		IF (left_groud_check1 AND left_groud_check2) THEN
			IF(head_f2 )THEN  ton_step4(in:=TRUE,pt:=T#1.5s);
			ELSE IF(head_b2 )THEN  ton_step4(in:=TRUE,pt:=T#1.0s);
			ELSE IF(head_b)THEN ton_step4(in:=TRUE,pt:=T#1.0s);
			ELSE IF(head_f)THEN ton_step4(in:=TRUE,pt:=T#2.0s);
			ELSE 	ton_step4(in:=TRUE,pt:=T#2.0s);
			END_IF
			END_IF
			END_IF
			END_IF
		END_IF


		IF ton1.q THEN leave_ground_sign:=1;ELSE leave_ground_sign:=0;END_IF
		IF( (ton_step4.q OR ton1.q )AND NOT level_second )OR (level_second AND ton4_second.Q )OR ton6_yanshi.Q THEN
			ton_step4(in:=0);
			ton1(in:=0);
			ton4_second(in:=0);
			extend_step:=5;
			step4_m1:=0;
			step4_m2:=0;
			step4_m3:=0;
			step4_m4:=0;
		END_IF
	END_IF

(*————————————————————————————自动支腿第五步————————————————————————————————————————*)
(*控制过程：精调平*)
	IF extend_step = 5 THEN
		tem2:=INT_TO_DINT(level_time)*1000;
		ton1(in:=1,pt:=DINT_TO_TIME(tem2));

		ton1();
		angle_x_real:=INT_TO_REAL(angle_x);
		angle_x_offset_real:=INT_TO_REAL(angle_x_offset);
		set_x:=REAL_TO_WORD(ABS(angle_x_real-angle_x_offset_real));
		angle_y_real:=INT_TO_REAL(angle_y);
		angle_y_offset_real:=INT_TO_REAL(angle_y_offset);
		set_y:=REAL_TO_WORD(ABS(angle_y_real-angle_y_offset_real));set_y := set_y*8/rl_ys;
		angle_ok_sign:=angle_ok/2;
		 IF REAL_TO_INT(ABS(angle_x_real-angle_x_offset_real)) <= angle_ok_sign THEN set_x := 0; END_IF;
		 IF REAL_TO_INT(ABS(angle_y_real-angle_y_offset_real)) <= angle_ok_sign THEN set_y := 0; END_IF;
(*--------------------------------------------------*)
		IF (angle_x-angle_x_offset)>=angle_ok_sign AND (angle_y-angle_y_offset)<=angle_ok_sign THEN
				left_front_desired:=set_x;
				right_back_desired:=set_y;
				left_back_desired:=set_x+set_y;
			IF NOT back_left_urt_ex_check THEN
				left_back_desired:=left_back_desired*2;left_front_desired:=left_front_desired/2;	right_back_desired:=right_back_desired/2;
    			END_IF
		ELSIF (angle_x-angle_x_offset)>=angle_ok_sign AND (angle_y-angle_y_offset)>=angle_ok_sign THEN
(*				right_front_desired:=set_y;*)
				left_back_desired:=set_x;
				left_front_desired:=set_x+set_y;
			IF NOT front_left_urt_ex_check THEN
				left_front_desired:=left_front_desired*2;	left_back_desired:=left_back_desired/2;	right_front_desired:=right_front_desired/2;
    			END_IF
		ELSIF (angle_x-angle_x_offset)<=angle_ok_sign AND (angle_y-angle_y_offset)<=angle_ok_sign THEN
				left_back_desired:=set_y;
				right_front_desired:=set_x;
				right_back_desired:=set_x+set_y;
			IF NOT back_right_urt_ex_check THEN
				right_back_desired:=right_back_desired*2;
				left_back_desired:=left_back_desired/2;
				right_front_desired:=right_front_desired/2;
    			END_IF
		ELSIF (angle_x-angle_x_offset)<=angle_ok_sign AND (angle_y-angle_y_offset)>=angle_ok_sign THEN
				right_back_desired:=set_x;
(*				left_front_desired:=set_y;*)
				right_front_desired:=set_x+set_y;
			IF NOT front_right_urt_ex_check THEN
				right_front_desired:=right_front_desired*2;	right_back_desired:=right_back_desired/2;	left_front_desired:=left_front_desired/2;
   			END_IF
		END_IF
(*************sl 增加******************s*)
			IF(head_b AND (angle_y>angle_y_offset))THEN
				IF(angle_x>angle_x_offset)THEN
						left_front_desired:=left_front_desired+20;
						right_front_desired:=right_front_desired+15;
						 left_back_desired:=REAL_TO_WORD(WORD_TO_REAL(left_back_desired)-5);
						 right_back_desired:=REAL_TO_WORD(WORD_TO_REAL(right_back_desired)-10);
				END_IF
				IF(angle_x<angle_x_offset)THEN
						left_front_desired:=left_front_desired+15;
						right_front_desired:=right_front_desired+20;
						left_back_desired:=REAL_TO_WORD(WORD_TO_REAL(left_back_desired)-10);
						 right_back_desired:=REAL_TO_WORD(WORD_TO_REAL(right_back_desired)-5);
				END_IF
			END_IF

			IF(head_f AND (angle_y<angle_y_offset))THEN
				IF(angle_x>angle_x_offset)THEN
						left_front_desired:=REAL_TO_WORD(WORD_TO_REAL(left_front_desired)-5);
						 right_front_desired:=REAL_TO_WORD(WORD_TO_REAL(right_front_desired)-10);
						left_back_desired:=left_back_desired+20;
						right_back_desired:=right_back_desired+15;
				END_IF
				IF(angle_x<angle_x_offset)THEN
						left_front_desired:=REAL_TO_WORD(WORD_TO_REAL(left_front_desired)-10);
						 right_front_desired:=REAL_TO_WORD(WORD_TO_REAL(right_front_desired)-5);
						left_back_desired:=left_back_desired+15;
						right_back_desired:=right_back_desired+20;
				END_IF
			END_IF
(*************sl 增加******************e*)
		IF NOT front_left_urt_ex_check1  THEN left_front_desired:=300;END_IF
		IF NOT back_left_urt_ex_check1   THEN  left_back_desired:=300;END_IF
		IF NOT front_right_urt_ex_check1 THEN   right_front_desired:=300;END_IF
		IF NOT back_right_urt_ex_check1 THEN  right_back_desired:=300;END_IF

IF (angle_y-angle_y_offset)<-step_4_limit+100 THEN left_front_desired:=0;right_front_desired:=0;END_IF
IF (angle_y-angle_y_offset)>step_4_limit-100 THEN right_back_desired:=0;left_back_desired:=0;END_IF
IF (angle_x-angle_x_offset)<-step_4_limit+100 THEN left_front_desired:=0;left_back_desired:=0;END_IF
IF (angle_x-angle_x_offset)>step_4_limit-100 THEN right_back_desired:=0;right_front_desired:=0;END_IF
		tontp(IN:= ABS(angle_x-angle_x_offset)<=angle_ok AND ABS(angle_y-angle_y_offset)<=angle_ok, PT:= T#200ms);
  (*精调平完成*)
		IF front_left_urt_ex_check AND front_right_urt_ex_check AND back_right_urt_ex_check AND back_left_urt_ex_check
			AND tontp.Q AND(( left_groud_check1 AND left_groud_check2)OR ton6_yanshi.Q  )THEN
(*			extend_do := 0;*)			ton1(in:=0);			(*leveled := 1;*)		alarmer_horn:=0;
			extend_step:=7;			down_valve_ctl:=0;
		END_IF;
		IF NOT(left_groud_check1 AND left_groud_check2)AND NOT ton6_yanshi.Q  THEN extend_step := 4; END_IF; (*有轮胎触地，回到撑起步骤*)
		IF ton1.q THEN ton1(in:=0); extend_step:=6;END_IF
	END_IF
(*————————————————————————————自动支腿第六步————————————————————————————————————————*)
	IF extend_step=6 THEN
		left_back_drawback_desired:=v_in_speed;
		left_front_drawback_desired:=v_in_speed;
		right_back_drawback_desired:=v_in_speed;
		right_front_drawback_desired:=v_in_speed;
		IF (NOT ton6_yanshi.Q AND (NOT left_groud_check1 OR NOT left_groud_check2)) OR
			NOT(front_left_urt_ex_check AND front_right_urt_ex_check AND back_left_urt_ex_check AND back_right_urt_ex_check) THEN
			extend_step:=4;
			ton6_yanshi(in:=0);
		END_IF
	END_IF

IF left_front_desired<0 OR  left_front_desired>10000 			THEN left_front_desired:=0;END_IF
IF left_back_desired<0 OR  left_back_desired>10000		 	THEN left_back_desired:=0;END_IF
IF right_front_desired<0 OR  right_front_desired>10000 		THEN right_front_desired:=0;END_IF
IF right_back_desired<0 OR  right_back_desired>10000		 THEN right_back_desired:=0;END_IF

(************************************伸支腿后展斗****************************************s*)
	stage_extend_do:=1;
	stage_draw_do:=0;

IF extend_step=7 THEN
	down_valve_ctl:=0;
	up_valve_ctl:=0;
	IF stage_extend_over THEN
		extend_do := 0;
		extend_step:=0;
		leveled := 1;
		alarmer_horn:=0;
		stage_extend_do:=0;
		stage_extend_over:=0;
	END_IF
END_IF
(************************************伸支腿后展斗****************************************e*)
ELSE
	extend_step:=0;
	stage_extend_do:=0;
	leave_ground_sign:=0;
END_IF



(*sl*****************************非正常调平判定*******************start*)
(**)
IF NOT auto_manu_choice AND((front_right_Lv_ex_check AND back_right_Lv_ex_check)OR(front_left_Lv_ex_check AND back_left_Lv_ex_check))AND front_left_urt_ex_check AND front_right_urt_ex_check AND back_left_urt_ex_check AND back_right_urt_ex_check AND ABS(angle_x-angle_x_offset)<=1.5*angle_ok AND ABS(angle_y-angle_y_offset)<=1.5*angle_ok THEN
	leveled:=1;
END_IF

(*sl*****************************非正常调平判定*******************end*)
(*
ton_second(in:=1,pt:=t#15s);
IF ton_second.Q  THEN allow_second:=1; END_IF
IF allow_second THEN
*)

(*
	IF NOT(front_left_urt_ex_check OR front_right_urt_ex_check OR back_left_urt_ex_check OR back_right_urt_ex_check)  AND  valve_act THEN
		leveled:=0;
	END_IF
ton_second()
*)
IF NOT(front_left_urt_ex_check OR front_right_urt_ex_check OR back_left_urt_ex_check OR back_right_urt_ex_check)  AND  valve_act THEN
	allow_second:=1;
ELSE
	allow_second:=0;
END_IF
ton_second(in:=allow_second,pt:=t#2s);
IF ton_second.Q THEN 		leveled:=0; 	ton_second(in:=0);	END_IF

(*————————————————————————————收支腿————————————————————————————————————————*)
(*收回支腿操作*)
auto_drawback_triger:=auto_drawback_triger_left OR auto_drawback_triger_right;
drawback_act(CLK:= auto_drawback_triger);
(*臂架到位而且不是第二次按收回旋钮*)
IF drawback_act.q  AND arm_to_station AND auto_manu_choice THEN
	withdraw_do:=(NOT withdraw_do);
	leave_ground_sign:=0;
	extend_do:=0;
	ton1(in:=0);ton6_yanshi(in:=0);
	withdraw_step:=100;
END_IF


(************************************收支腿前翻斗****************************************e*)

(*收回步骤1：收垂直腿*)
IF withdraw_do THEN

(************************************收支腿前翻斗****************************************s*)
(*
IF withdraw_step=10 THEN
	stage_extend_do:=0;
	stage_draw_do:=1;
	down_valve_ctl:=0;
	up_valve_ctl:=1;
	IF stage_draw_over THEN
		withdraw_step:=100;
		stage_draw_do:=0;
		stage_draw_over:=0;
	END_IF
ELSE
	stage_draw_do:=0;
END_IF
*)
stage_extend_do:=0;
stage_draw_do:=1;
IF stage_draw_over THEN
	stage_draw_do:=0;
	stage_draw_over:=0;
END_IF


IF withdraw_step=100 THEN
	ton_withdraw(in:=1,pt:=t#1s);
	IF(ton_withdraw.Q)THEN
		withdraw_step:=1;
		ton_withdraw(in:=0);
	END_IF
END_IF

	alarmer_horn:=1;

	IF withdraw_step=1 THEN
		tem2:=INT_TO_DINT(v_in_time)*1000;
		ton1(in:=1,pt:=DINT_TO_TIME(tem2));
		ton1();
		IF NOT front_left_urt_drb_check 		THEN left_front_drawback_desired:=v_in_speed; 	ELSE	left_front_drawback_desired:=0;		END_IF
		IF NOT front_right_urt_drb_check 	THEN right_front_drawback_desired:=v_in_speed;	ELSE	right_front_drawback_desired:=0; 	END_IF
		IF NOT back_left_urt_drb_check 		THEN left_back_drawback_desired:=v_in_speed; 	ELSE	left_back_drawback_desired:=0;		END_IF
		IF NOT back_right_urt_drb_check	THEN right_back_drawback_desired:=v_in_speed; ELSE	right_back_drawback_desired:=0;	END_IF

(*************sl 增加******************s*结合象限角结合XY变化率来对速度开口进行加减*)
IF(NOT  left_groud_check1 AND NOT  left_groud_check2)THEN
	withdraw_t1(in:=1,pt:=t#2s);
	IF(withdraw_t1.Q)THEN
		withdraw_m5:=1;
	END_IF
END_IF

IF(NOT withdraw_m5 )OR(head_b2 AND(back_right_urt_ex_check OR back_left_urt_ex_check))OR(head_f2 AND(front_right_urt_ex_check OR front_left_urt_ex_check))THEN
	IF  NOT( angle_withdraw_x1=angle_x )THEN
		angle_withdraw_x2:=angle_withdraw_x1;
		angle_withdraw_x1:=angle_x;
	END_IF
	IF  NOT( angle_withdraw_y1=angle_y )THEN
		angle_withdraw_y2:=angle_withdraw_y1;
		angle_withdraw_y1:=angle_y;
	END_IF
	withdraw_mx:=angle_withdraw_x1-angle_withdraw_x2;
	withdraw_my:=angle_withdraw_y1-angle_withdraw_y2;

	CASE angle_dir OF(*清零 以及 各项先+-50*)
		1:
			withdraw_m1:=1;
			IF(withdraw_m2 OR withdraw_m3 OR withdraw_m4)THEN
				withdraw_fl:=0;
				withdraw_fr:=0;
				withdraw_bl:=0;
				withdraw_br:=0;
				withdraw_m2:=0;withdraw_m3:=0;withdraw_m4:=0;
			END_IF
			IF(angle_x>=angle_x_offset+50)THEN
				IF(withdraw_mx>0)THEN withdraw_fr:=withdraw_fr+w_value; withdraw_br:=withdraw_br+w_value;   END_IF
			END_IF
			IF(angle_y<=angle_y_offset-50)THEN
				 withdraw_fl:=withdraw_fl+w_value;  withdraw_fr:=withdraw_fr+w_value;
			END_IF
			IF(withdraw_my<0)THEN
				withdraw_fl:=withdraw_fl+w_value;  withdraw_fr:=withdraw_fr+w_value;
			END_IF

		2:
			withdraw_m2:=1;
			IF(withdraw_m1 OR withdraw_m3 OR withdraw_m4)THEN
				withdraw_fl:=0;
				withdraw_fr:=0;
				withdraw_bl:=0;
				withdraw_br:=0;
				withdraw_m1:=0;withdraw_m3:=0;withdraw_m4:=0;
			END_IF
			IF(angle_x>=angle_x_offset+50)THEN
				IF(withdraw_mx>0)THEN withdraw_fr:=withdraw_fr+w_value; withdraw_br:=withdraw_br+w_value;   END_IF
			END_IF
			IF(angle_y>=angle_y_offset+50)THEN
				 withdraw_bl:=withdraw_bl+w_value;  withdraw_br:=withdraw_br+w_value;
			END_IF
			IF(withdraw_my>0)THEN
				withdraw_bl:=withdraw_bl+w_value;  withdraw_br:=withdraw_br+w_value;
			END_IF
		3:
			withdraw_m3:=1;
			IF(withdraw_m2 OR withdraw_m1 OR withdraw_m4)THEN
				withdraw_fl:=0;
				withdraw_fr:=0;
				withdraw_bl:=0;
				withdraw_br:=0;
				withdraw_m1:=0;withdraw_m2:=0;withdraw_m4:=0;
			END_IF
			IF(angle_x<=angle_x_offset-50)THEN
				IF(withdraw_mx<0)THEN withdraw_fl:=withdraw_fl+w_value; withdraw_bl:=withdraw_bl+w_value;   END_IF
			END_IF
			IF(angle_y<=angle_y_offset-50)THEN
				 withdraw_fl:=withdraw_fl+w_value;  withdraw_fr:=withdraw_fr+w_value;
			END_IF
			IF(withdraw_my<0)THEN
				withdraw_fl:=withdraw_fl+w_value;  withdraw_fr:=withdraw_fr+w_value;
			END_IF
		4:
			withdraw_m4:=1;
			IF(withdraw_m2 OR withdraw_m3 OR withdraw_m1)THEN
				withdraw_fl:=0;
				withdraw_fr:=0;
				withdraw_bl:=0;
				withdraw_br:=0;
				withdraw_m1:=0;withdraw_m2:=0;withdraw_m3:=0;
			END_IF
			IF(angle_x<=angle_x_offset-50)THEN
				IF(withdraw_mx<0)THEN withdraw_fl:=withdraw_fl+w_value; withdraw_bl:=withdraw_bl+w_value;   		END_IF
			END_IF
			IF(angle_y>=angle_y_offset+50)THEN
				withdraw_bl:=withdraw_bl+w_value;  withdraw_br:=withdraw_br+w_value;
			END_IF
			IF(withdraw_my>0)THEN
				withdraw_bl:=withdraw_bl+w_value;  withdraw_br:=withdraw_br+w_value;
			END_IF
	END_CASE

		IF NOT front_left_urt_drb_check 		THEN left_front_drawback_desired:=v_in_speed-withdraw_fl; 			ELSE	left_front_drawback_desired:=0;		END_IF
		IF NOT front_right_urt_drb_check 	THEN right_front_drawback_desired:=v_in_speed-withdraw_fr;		ELSE	right_front_drawback_desired:=0; 	END_IF
		IF NOT back_left_urt_drb_check 		THEN left_back_drawback_desired:=v_in_speed-withdraw_bl; 		ELSE	left_back_drawback_desired:=0;		END_IF
		IF NOT back_right_urt_drb_check	THEN right_back_drawback_desired:=v_in_speed-withdraw_br;	 	ELSE	right_back_drawback_desired:=0;	END_IF
ELSE
		withdraw_fl:=0;
		withdraw_fr:=0;
		withdraw_bl:=0;
		withdraw_br:=0;
END_IF
(*************sl 增加******************e*)

		IF (front_left_urt_drb_check AND front_right_urt_drb_check AND back_left_urt_drb_check AND back_right_urt_drb_check)OR ton1.q THEN
		ton1(in:=0);
		withdraw_t1(in:=0);
		withdraw_step:=2;
		withdraw_m5:=0;
		END_IF

	END_IF
	IF withdraw_step=2 THEN

		tem2:=INT_TO_DINT(v_in_time)*1000;
		ton1(in:=1,pt:=DINT_TO_TIME(tem2));
		ton1();
		IF NOT front_left_Lv_drb_check  	THEN left_front_lv_drb_valve:=1;   	ELSE	left_front_lv_drb_valve:=0;	END_IF
		IF NOT back_left_lv_drb_check   	THEN left_back_lv_drb_valve:=1;		ELSE	left_back_lv_drb_valve:=0; 	END_IF
		IF NOT front_right_lv_drb_check 	THEN right_front_lv_drb_valve:=1; 	ELSE	right_front_lv_drb_valve:=0;	END_IF
		IF NOT back_right_lv_drb_check  THEN right_back_lv_drb_valve:=1; 	ELSE	right_back_lv_drb_valve:=0;	END_IF
		IF ((front_left_Lv_drb_check AND back_left_lv_drb_check AND front_right_lv_drb_check AND back_right_lv_drb_check) OR ton1.q )AND NOT stage_draw_do THEN
			ton1(in:=0);
			withdraw_do:=0;
			withdraw_step:=0;
			down_valve_ctl:=0;
			up_valve_ctl:=0;
			head_f:=0;head_b:=0;head_f2:=0;head_b2:=0;side_l:=0;side_r:=0;
		END_IF
END_IF
	IF NOT front_left_urt_drb_check 		THEN left_front_drawback_desired:=v_in_speed; 	ELSE	left_front_drawback_desired:=0;				END_IF
			IF NOT front_right_urt_drb_check 	THEN right_front_drawback_desired:=v_in_speed;	ELSE	right_front_drawback_desired:=0; 	END_IF
			IF NOT back_left_urt_drb_check 		THEN left_back_drawback_desired:=v_in_speed; 	ELSE	left_back_drawback_desired:=0;		END_IF
			IF NOT back_right_urt_drb_check	THEN right_back_drawback_desired:=v_in_speed; ELSE	right_back_drawback_desired:=0;	END_IF
	END_IF

IF withdraw_do THEN
	leveled:=0;
ELSE
	withdraw_step:=0;
	stage_draw_do:=0;
END_IF
END_PROGRAM

(* POU TRIGER_Regulation/LEVEL_PROMPT, ST *)
PROGRAM LEVEL_PROMPT
VAR
	left_front_desired_prom_add1: BOOL;
	R_TRIG1: R_TRIG;
	R_TRIG2: R_TRIG;
	R_TRIG3: R_TRIG;
	R_TRIG4: R_TRIG;
	R_TRIG5: R_TRIG;
	R_TRIG6: R_TRIG;
	R_TRIG7: R_TRIG;
	R_TRIG8: R_TRIG;


	R_TRIG9: R_TRIG;
	R_TRIG10: R_TRIG;
	R_TRIG11: R_TRIG;
	R_TRIG12: R_TRIG;
	R_TRIG13: R_TRIG;
	R_TRIG14: R_TRIG;
	R_TRIG15: R_TRIG;
	R_TRIG16: R_TRIG;


	R_TRIG17: R_TRIG;
	R_TRIG18: R_TRIG;
	R_TRIG19: R_TRIG;
	R_TRIG20: R_TRIG;
	R_TRIG21: R_TRIG;
	R_TRIG22: R_TRIG;
	R_TRIG23: R_TRIG;
	R_TRIG24: R_TRIG;

	fl_o_fac_b1: BOOL;
	fr_o_fac_b1: BOOL;
	rl_o_fac_b1: BOOL;
	rr_o_fac_b1: BOOL;
	fl_i_fac_b1: BOOL;
	fr_i_fac_b1: BOOL;
	rl_i_fac_b1: BOOL;
	rr_i_fac_b1: BOOL;

	fl_o_fac_b_l1: BOOL;
	fr_o_fac_b_l1: BOOL;
	rl_o_fac_b_l1: BOOL;
	rr_o_fac_b_l1: BOOL;
	fl_i_fac_b_l1: BOOL;
	fr_i_fac_b_l1: BOOL;
	rl_i_fac_b_l1: BOOL;
	rr_i_fac_b_l1: BOOL;

	fl_o_fac_b_r1: BOOL;
	fr_o_fac_b_r1: BOOL;
	rl_o_fac_b_r1: BOOL;
	rr_o_fac_b_r1: BOOL;
	fl_i_fac_b_r1: BOOL;
	fr_i_fac_b_r1: BOOL;
	rl_i_fac_b_r1: BOOL;
	rr_i_fac_b_r1: BOOL;


END_VAR
digit_data_in_cylinder();

IF(head_b2)OR(head_f2)THEN
	case_curve2();
ELSE
	case_curve();
END_IF


IF NOT ramp_selected THEN

	analog_in_out_cylinder();

	R_TRIG1(CLK:=fl_o_fac_b , Q=>fl_o_fac_b1 );
	R_TRIG2(CLK:=fl_i_fac_b , Q=>fl_i_fac_b1 );
	IF fl_o_fac_b1 THEN fl_fac_nr:=fl_fac_nr+1;END_IF
	IF fl_i_fac_b1 THEN fl_fac_nr:=fl_fac_nr-1;END_IF
	IF fl_fac_nr>10 THEN fl_fac_nr:=10;END_IF
	IF fl_fac_nr<-10 THEN fl_fac_nr:=-10;END_IF

	R_TRIG3(CLK:=fl_o_fac_b_l , Q=>fl_o_fac_b_l1 );
	R_TRIG4(CLK:=fl_i_fac_b_l , Q=>fl_i_fac_b_l1 );
	IF fl_o_fac_b_l1 THEN fl_fac_l_nr:=fl_fac_l_nr+1;END_IF
	IF fl_i_fac_b_l1 THEN fl_fac_l_nr:=fl_fac_l_nr-1;END_IF
	IF fl_fac_l_nr>10 THEN fl_fac_l_nr:=10;END_IF
	IF fl_fac_l_nr<-10 THEN fl_fac_l_nr:=-10;END_IF

	R_TRIG5(CLK:=fl_o_fac_b_r , Q=>fl_o_fac_b_r1 );
	R_TRIG6(CLK:=fl_i_fac_b_r , Q=>fl_i_fac_b_r1 );
	IF fl_o_fac_b_r1 THEN fl_fac_r_nr:=fl_fac_r_nr+1;END_IF
	IF fl_i_fac_b_r1 THEN fl_fac_r_nr:=fl_fac_r_nr-1;END_IF
	IF fl_fac_r_nr>10 THEN fl_fac_r_nr:=10;END_IF
	IF fl_fac_r_nr<-10 THEN fl_fac_r_nr:=-10;END_IF
	(***********************************)

	R_TRIG7(CLK:=fr_o_fac_b , Q=>fr_o_fac_b1 );
	R_TRIG8(CLK:=fr_i_fac_b , Q=>fr_i_fac_b1 );
	IF fr_o_fac_b1 THEN fr_fac_nr:=fr_fac_nr+1;END_IF
	IF fr_i_fac_b1 THEN fr_fac_nr:=fr_fac_nr-1;END_IF
	IF fr_fac_nr>10 THEN fr_fac_nr:=10;END_IF
	IF fr_fac_nr<-10 THEN fr_fac_nr:=-10;END_IF

	R_TRIG9(CLK:=fr_o_fac_b_l , Q=>fr_o_fac_b_l1 );
	R_TRIG10(CLK:=fr_i_fac_b_l , Q=>fr_i_fac_b_l1 );
	IF fr_o_fac_b_l1 THEN fr_fac_l_nr:=fr_fac_l_nr+1;END_IF
	IF fr_i_fac_b_l1 THEN fr_fac_l_nr:=fr_fac_l_nr-1;END_IF
	IF fr_fac_l_nr>10 THEN fr_fac_l_nr:=10;END_IF
	IF fr_fac_l_nr<-10 THEN fr_fac_l_nr:=-10;END_IF

	R_TRIG11(CLK:=fr_o_fac_b_r , Q=>fr_o_fac_b_r1 );
	R_TRIG12(CLK:=fr_i_fac_b_r , Q=>fr_i_fac_b_r1 );
	IF fr_o_fac_b_r1 THEN fr_fac_r_nr:=fr_fac_r_nr+1;END_IF
	IF fr_i_fac_b_r1 THEN fr_fac_r_nr:=fr_fac_r_nr-1;END_IF
	IF fr_fac_r_nr>10 THEN fr_fac_r_nr:=10;END_IF
	IF fr_fac_r_nr<-10 THEN fr_fac_r_nr:=-10;END_IF

	(*******************************)

	R_TRIG13(CLK:=rl_o_fac_b , Q=>rl_o_fac_b1 );
	R_TRIG14(CLK:=rl_i_fac_b , Q=>rl_i_fac_b1 );
	IF rl_o_fac_b1 THEN rl_fac_nr:=rl_fac_nr+1;END_IF
	IF rl_i_fac_b1 THEN rl_fac_nr:=rl_fac_nr-1;END_IF
	IF rl_fac_nr>10 THEN rl_fac_nr:=10;END_IF
	IF rl_fac_nr<-10 THEN rl_fac_nr:=-10;END_IF

	R_TRIG15(CLK:=rl_o_fac_b_l , Q=>rl_o_fac_b_l1 );
	R_TRIG16(CLK:=rl_i_fac_b_l , Q=>rl_i_fac_b_l1 );
	IF rl_o_fac_b_l1 THEN rl_fac_l_nr:=rl_fac_l_nr+1;END_IF
	IF rl_i_fac_b_l1 THEN rl_fac_l_nr:=rl_fac_l_nr-1;END_IF
	IF rl_fac_l_nr>10 THEN rl_fac_l_nr:=10;END_IF
	IF rl_fac_l_nr<-10 THEN rl_fac_l_nr:=-10;END_IF

	R_TRIG17(CLK:=rl_o_fac_b_r , Q=>rl_o_fac_b_r1 );
	R_TRIG18(CLK:=rl_i_fac_b_r , Q=>rl_i_fac_b_r1 );
	IF rl_o_fac_b_r1 THEN rl_fac_r_nr:=rl_fac_r_nr+1;END_IF
	IF rl_i_fac_b_r1 THEN rl_fac_r_nr:=rl_fac_r_nr-1;END_IF
	IF rl_fac_r_nr>10 THEN rl_fac_r_nr:=10;END_IF
	IF rl_fac_r_nr<-10 THEN rl_fac_r_nr:=-10;END_IF

	(**************************)

	R_TRIG19(CLK:=rr_o_fac_b , Q=>rr_o_fac_b1 );
	R_TRIG20(CLK:=rr_i_fac_b , Q=>rr_i_fac_b1 );
	IF rr_o_fac_b1 THEN rr_fac_nr:=rr_fac_nr+1;END_IF
	IF rr_i_fac_b1 THEN rr_fac_nr:=rr_fac_nr-1;END_IF
	IF rr_fac_nr>10 THEN rr_fac_nr:=10;END_IF
	IF rr_fac_nr<-10 THEN rr_fac_nr:=-10;END_IF

	R_TRIG21(CLK:=rr_o_fac_b_l , Q=>rr_o_fac_b_l1 );
	R_TRIG22(CLK:=rr_i_fac_b_l , Q=>rr_i_fac_b_l1 );
	IF rr_o_fac_b_l1 THEN rr_fac_l_nr:=rr_fac_l_nr+1;END_IF
	IF rr_i_fac_b_l1 THEN rr_fac_l_nr:=rr_fac_l_nr-1;END_IF
	IF rr_fac_l_nr>10 THEN rr_fac_l_nr:=10;END_IF
	IF rr_fac_l_nr<-10 THEN rr_fac_l_nr:=-10;END_IF

	R_TRIG23(CLK:=rr_o_fac_b_r , Q=>rr_o_fac_b_r1 );
	R_TRIG24(CLK:=rr_i_fac_b_r , Q=>rr_i_fac_b_r1 );
	IF rr_o_fac_b_r1 THEN rr_fac_r_nr:=rr_fac_r_nr+1;END_IF
	IF rr_i_fac_b_r1 THEN rr_fac_r_nr:=rr_fac_r_nr-1;END_IF
	IF rr_fac_r_nr>10 THEN rr_fac_r_nr:=10;END_IF
	IF rr_fac_r_nr<-10 THEN rr_fac_r_nr:=-10;END_IF

ELSE

	analog_in_out_cylinder2();

	R_TRIG1(CLK:=fl_o_fac_b , Q=>fl_o_fac_b1 );
	R_TRIG2(CLK:=fl_i_fac_b , Q=>fl_i_fac_b1 );
	IF fl_o_fac_b1 THEN fl_fac_nr2:=fl_fac_nr2+1;END_IF
	IF fl_i_fac_b1 THEN fl_fac_nr2:=fl_fac_nr2-1;END_IF
	IF fl_fac_nr>10 THEN fl_fac_nr2:=10;END_IF
	IF fl_fac_nr<-10 THEN fl_fac_nr2:=-10;END_IF

	R_TRIG3(CLK:=fl_o_fac_b_l , Q=>fl_o_fac_b_l1 );
	R_TRIG4(CLK:=fl_i_fac_b_l , Q=>fl_i_fac_b_l1 );
	IF fl_o_fac_b_l1 THEN fl_fac_l_nr2:=fl_fac_l_nr2+1;END_IF
	IF fl_i_fac_b_l1 THEN fl_fac_l_nr2:=fl_fac_l_nr2-1;END_IF
	IF fl_fac_l_nr>10 THEN fl_fac_l_nr2:=10;END_IF
	IF fl_fac_l_nr<-10 THEN fl_fac_l_nr2:=-10;END_IF

	R_TRIG5(CLK:=fl_o_fac_b_r , Q=>fl_o_fac_b_r1 );
	R_TRIG6(CLK:=fl_i_fac_b_r , Q=>fl_i_fac_b_r1 );
	IF fl_o_fac_b_r1 THEN fl_fac_r_nr2:=fl_fac_r_nr2+1;END_IF
	IF fl_i_fac_b_r1 THEN fl_fac_r_nr2:=fl_fac_r_nr2-1;END_IF
	IF fl_fac_r_nr>10 THEN fl_fac_r_nr2:=10;END_IF
	IF fl_fac_r_nr<-10 THEN fl_fac_r_nr2:=-10;END_IF
	(***********************************)

	R_TRIG7(CLK:=fr_o_fac_b , Q=>fr_o_fac_b1 );
	R_TRIG8(CLK:=fr_i_fac_b , Q=>fr_i_fac_b1 );
	IF fr_o_fac_b1 THEN fr_fac_nr2:=fr_fac_nr2+1;END_IF
	IF fr_i_fac_b1 THEN fr_fac_nr2:=fr_fac_nr2-1;END_IF
	IF fr_fac_nr>10 THEN fr_fac_nr2:=10;END_IF
	IF fr_fac_nr<-10 THEN fr_fac_nr2:=-10;END_IF

	R_TRIG9(CLK:=fr_o_fac_b_l , Q=>fr_o_fac_b_l1 );
	R_TRIG10(CLK:=fr_i_fac_b_l , Q=>fr_i_fac_b_l1 );
	IF fr_o_fac_b_l1 THEN fr_fac_l_nr2:=fr_fac_l_nr2+1;END_IF
	IF fr_i_fac_b_l1 THEN fr_fac_l_nr2:=fr_fac_l_nr2-1;END_IF
	IF fr_fac_l_nr>10 THEN fr_fac_l_nr2:=10;END_IF
	IF fr_fac_l_nr<-10 THEN fr_fac_l_nr2:=-10;END_IF

	R_TRIG11(CLK:=fr_o_fac_b_r , Q=>fr_o_fac_b_r1 );
	R_TRIG12(CLK:=fr_i_fac_b_r , Q=>fr_i_fac_b_r1 );
	IF fr_o_fac_b_r1 THEN fr_fac_r_nr2:=fr_fac_r_nr2+1;END_IF
	IF fr_i_fac_b_r1 THEN fr_fac_r_nr2:=fr_fac_r_nr2-1;END_IF
	IF fr_fac_r_nr>10 THEN fr_fac_r_nr2:=10;END_IF
	IF fr_fac_r_nr<-10 THEN fr_fac_r_nr2:=-10;END_IF

	(*******************************)

	R_TRIG13(CLK:=rl_o_fac_b , Q=>rl_o_fac_b1 );
	R_TRIG14(CLK:=rl_i_fac_b , Q=>rl_i_fac_b1 );
	IF rl_o_fac_b1 THEN rl_fac_nr2:=rl_fac_nr2+1;END_IF
	IF rl_i_fac_b1 THEN rl_fac_nr2:=rl_fac_nr2-1;END_IF
	IF rl_fac_nr>10 THEN rl_fac_nr2:=10;END_IF
	IF rl_fac_nr<-10 THEN rl_fac_nr2:=-10;END_IF

	R_TRIG15(CLK:=rl_o_fac_b_l , Q=>rl_o_fac_b_l1 );
	R_TRIG16(CLK:=rl_i_fac_b_l , Q=>rl_i_fac_b_l1 );
	IF rl_o_fac_b_l1 THEN rl_fac_l_nr2:=rl_fac_l_nr2+1;END_IF
	IF rl_i_fac_b_l1 THEN rl_fac_l_nr2:=rl_fac_l_nr2-1;END_IF
	IF rl_fac_l_nr>10 THEN rl_fac_l_nr2:=10;END_IF
	IF rl_fac_l_nr<-10 THEN rl_fac_l_nr2:=-10;END_IF

	R_TRIG17(CLK:=rl_o_fac_b_r , Q=>rl_o_fac_b_r1 );
	R_TRIG18(CLK:=rl_i_fac_b_r , Q=>rl_i_fac_b_r1 );
	IF rl_o_fac_b_r1 THEN rl_fac_r_nr2:=rl_fac_r_nr2+1;END_IF
	IF rl_i_fac_b_r1 THEN rl_fac_r_nr2:=rl_fac_r_nr2-1;END_IF
	IF rl_fac_r_nr>10 THEN rl_fac_r_nr2:=10;END_IF
	IF rl_fac_r_nr<-10 THEN rl_fac_r_nr2:=-10;END_IF

	(**************************)

	R_TRIG19(CLK:=rr_o_fac_b , Q=>rr_o_fac_b1 );
	R_TRIG20(CLK:=rr_i_fac_b , Q=>rr_i_fac_b1 );
	IF rr_o_fac_b1 THEN rr_fac_nr2:=rr_fac_nr2+1;END_IF
	IF rr_i_fac_b1 THEN rr_fac_nr2:=rr_fac_nr2-1;END_IF
	IF rr_fac_nr>10 THEN rr_fac_nr2:=10;END_IF
	IF rr_fac_nr<-10 THEN rr_fac_nr2:=-10;END_IF

	R_TRIG21(CLK:=rr_o_fac_b_l , Q=>rr_o_fac_b_l1 );
	R_TRIG22(CLK:=rr_i_fac_b_l , Q=>rr_i_fac_b_l1 );
	IF rr_o_fac_b_l1 THEN rr_fac_l_nr2:=rr_fac_l_nr2+1;END_IF
	IF rr_i_fac_b_l1 THEN rr_fac_l_nr2:=rr_fac_l_nr2-1;END_IF
	IF rr_fac_l_nr>10 THEN rr_fac_l_nr2:=10;END_IF
	IF rr_fac_l_nr<-10 THEN rr_fac_l_nr2:=-10;END_IF

	R_TRIG23(CLK:=rr_o_fac_b_r , Q=>rr_o_fac_b_r1 );
	R_TRIG24(CLK:=rr_i_fac_b_r , Q=>rr_i_fac_b_r1 );
	IF rr_o_fac_b_r1 THEN rr_fac_r_nr2:=rr_fac_r_nr2+1;END_IF
	IF rr_i_fac_b_r1 THEN rr_fac_r_nr2:=rr_fac_r_nr2-1;END_IF
	IF rr_fac_r_nr>10 THEN rr_fac_r_nr2:=10;END_IF
	IF rr_fac_r_nr<-10 THEN rr_fac_r_nr2:=-10;END_IF


END_IF
END_PROGRAM

(* POU TRIGER_Regulation/digit_data_in_cylinder, FBD *)
PROGRAM digit_data_in_cylinder
VAR


	P_31_0:UNPACK;
	P_31_1:UNPACK;
	P_31_2:UNPACK;
	P_31_3:UNPACK;



END_VAR
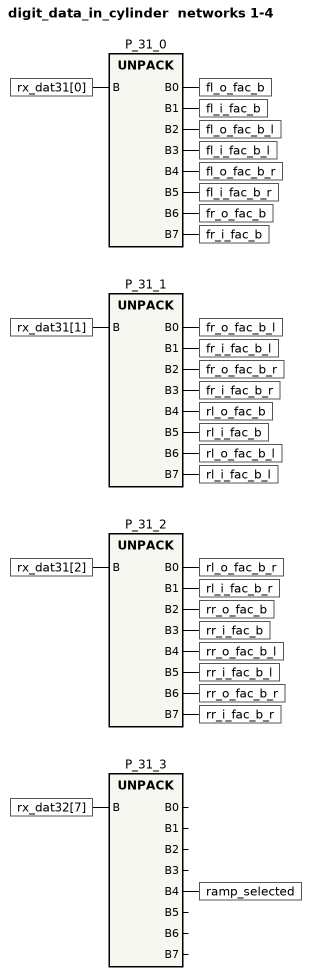
_FBD_ (* Function Block Diagram *)
NETWORK 1
	P_31_0:UNPACK(B: rx_dat31[0], B1 => fl_i_fac_b, B2 => fl_o_fac_b_l, B3 => fl_i_fac_b_l, B4 => fl_o_fac_b_r, B5 => fl_i_fac_b_r, B6 => fr_o_fac_b, B7 => fr_i_fac_b) => fl_o_fac_b
NETWORK 2
	P_31_1:UNPACK(B: rx_dat31[1], B1 => fr_i_fac_b_l, B2 => fr_o_fac_b_r, B3 => fr_i_fac_b_r, B4 => rl_o_fac_b, B5 => rl_i_fac_b, B6 => rl_o_fac_b_l, B7 => rl_i_fac_b_l) => fr_o_fac_b_l
NETWORK 3
	P_31_2:UNPACK(B: rx_dat31[2], B1 => rl_i_fac_b_r, B2 => rr_o_fac_b, B3 => rr_i_fac_b, B4 => rr_o_fac_b_l, B5 => rr_i_fac_b_l, B6 => rr_o_fac_b_r, B7 => rr_i_fac_b_r) => rl_o_fac_b_r
NETWORK 4
	P_31_3:UNPACK(B: rx_dat32[7], B4 => ramp_selected)
_END_FBD_
(* the same logic as Structured Text *)
(* Network 1 *)
P_31_0(B := rx_dat31[0]);
fl_i_fac_b := P_31_0.B1;
fl_o_fac_b_l := P_31_0.B2;
fl_i_fac_b_l := P_31_0.B3;
fl_o_fac_b_r := P_31_0.B4;
fl_i_fac_b_r := P_31_0.B5;
fr_o_fac_b := P_31_0.B6;
fr_i_fac_b := P_31_0.B7;
fl_o_fac_b := P_31_0.B0;
(* Network 2 *)
P_31_1(B := rx_dat31[1]);
fr_i_fac_b_l := P_31_1.B1;
fr_o_fac_b_r := P_31_1.B2;
fr_i_fac_b_r := P_31_1.B3;
rl_o_fac_b := P_31_1.B4;
rl_i_fac_b := P_31_1.B5;
rl_o_fac_b_l := P_31_1.B6;
rl_i_fac_b_l := P_31_1.B7;
fr_o_fac_b_l := P_31_1.B0;
(* Network 3 *)
P_31_2(B := rx_dat31[2]);
rl_i_fac_b_r := P_31_2.B1;
rr_o_fac_b := P_31_2.B2;
rr_i_fac_b := P_31_2.B3;
rr_o_fac_b_l := P_31_2.B4;
rr_i_fac_b_l := P_31_2.B5;
rr_o_fac_b_r := P_31_2.B6;
rr_i_fac_b_r := P_31_2.B7;
rl_o_fac_b_r := P_31_2.B0;
(* Network 4 *)
P_31_3(B := rx_dat32[7]);
ramp_selected := P_31_3.B4;
END_PROGRAM

(* POU TRIGER_Regulation/case_curve2, ST *)
PROGRAM case_curve2
VAR

	right_temp: BOOL;
	test_result: INT;
	left_temp: BOOL;


	array_cc: ARRAY[0..20]OF cc_point;
	cc_0:ARRAY[0..10] OF POINT       :=(X:=0,Y:=0),(X:=1,Y:=100),  (X:=500,Y:=200), (X:=1000,Y:=220), 7((X:=1000,Y:=520));
	cc_1:ARRAY[0..10] OF POINT       :=(X:=0,Y:=0),(X:=1,Y:=100),  (X:=500,Y:=220), (X:=1000,Y:=240), 7((X:=1000,Y:=520));
	cc_2:ARRAY[0..10] OF POINT       :=(X:=0,Y:=0),(X:=1,Y:=100),  (X:=500,Y:=240), (X:=1000,Y:=260), 7((X:=1000,Y:=520));
	cc_3:ARRAY[0..10] OF POINT       :=(X:=0,Y:=0),(X:=1,Y:=120),  (X:=500,Y:=260), (X:=1000,Y:=300), 7((X:=1000,Y:=520));
	cc_4:ARRAY[0..10] OF POINT       :=(X:=0,Y:=0),(X:=1,Y:=140),  (X:=500,Y:=280), (X:=1000,Y:=320), 7((X:=1000,Y:=520));
	cc_5:ARRAY[0..10] OF POINT       :=(X:=0,Y:=0),(X:=1,Y:=160),  (X:=500,Y:=300), (X:=1000,Y:=340), 7((X:=1000,Y:=520));
	cc_6:ARRAY[0..10] OF POINT       :=(X:=0,Y:=0),(X:=1,Y:=180),  (X:=500,Y:=320), (X:=1000,Y:=360), 7((X:=1000,Y:=520));
	cc_7:ARRAY[0..10] OF POINT       :=(X:=0,Y:=0),(X:=1,Y:=200),  (X:=500,Y:=360), (X:=1000,Y:=400), 7((X:=1000,Y:=520));
	cc_8:ARRAY[0..10] OF POINT       :=(X:=0,Y:=0),(X:=1,Y:=220),  (X:=500,Y:=400), (X:=1000,Y:=440), 7((X:=1000,Y:=520));
	cc_9:ARRAY[0..10] OF POINT       :=(X:=0,Y:=0),(X:=1,Y:=240),  (X:=500,Y:=460), (X:=1000,Y:=480), 7((X:=1000,Y:=520));
	cc_10:ARRAY[0..10] OF POINT       :=(X:=0,Y:=0),(X:=1,Y:=260),  (X:=500,Y:=480), (X:=1000,Y:=520), 7((X:=1000,Y:=520));(*常规启动电流，对应常规支腿速度*)
	cc_11:ARRAY[0..10] OF POINT       :=(X:=0,Y:=0),(X:=1,Y:=280),  (X:=500,Y:=480), (X:=1000,Y:=520), 7((X:=1000,Y:=520));
	cc_12:ARRAY[0..10] OF POINT       :=(X:=0,Y:=0),(X:=1,Y:=280),  (X:=500,Y:=500), (X:=1000,Y:=540), 7((X:=1000,Y:=520));
	cc_13:ARRAY[0..10] OF POINT       :=(X:=0,Y:=0),(X:=1,Y:=300),  (X:=500,Y:=500), (X:=1000,Y:=540), 7((X:=1000,Y:=520));
	cc_14:ARRAY[0..10] OF POINT       :=(X:=0,Y:=0),(X:=1,Y:=300),  (X:=500,Y:=520), (X:=1000,Y:=560), 7((X:=1000,Y:=520));
	cc_15:ARRAY[0..10] OF POINT       :=(X:=0,Y:=0),(X:=1,Y:=320),  (X:=500,Y:=520), (X:=1000,Y:=560), 7((X:=1000,Y:=520));
	cc_16:ARRAY[0..10] OF POINT       :=(X:=0,Y:=0),(X:=1,Y:=320),  (X:=500,Y:=540), (X:=1000,Y:=580), 7((X:=1000,Y:=520));
	cc_17:ARRAY[0..10] OF POINT       :=(X:=0,Y:=0),(X:=1,Y:=340),  (X:=500,Y:=540), (X:=1000,Y:=580), 7((X:=1000,Y:=520));
	cc_18:ARRAY[0..10] OF POINT       :=(X:=0,Y:=0),(X:=1,Y:=360),  (X:=500,Y:=540), (X:=1000,Y:=580), 7((X:=1000,Y:=520));
	cc_19:ARRAY[0..10] OF POINT       :=(X:=0,Y:=0),(X:=1,Y:=360),  (X:=500,Y:=560), (X:=1000,Y:=600), 7((X:=1000,Y:=520));
	cc_20:ARRAY[0..10] OF POINT       :=(X:=0,Y:=0),(X:=1,Y:=400),  (X:=500,Y:=600), (X:=1000,Y:=700), 7((X:=1000,Y:=520));
	fl_A1: CHARCURVE;
	fr_A1: CHARCURVE;
	rl_A1: CHARCURVE;
	rr_A1: CHARCURVE;
	left_front_desired_temp: WORD;



	left_front_desired_CR0032_temp										: WORD;(*左前垂直伸*)
	right_front_desired_CR0032_temp								: WORD;(*右前垂直伸*)
	left_back_desired_CR0032_temp										: WORD;(*左后垂直伸*)
	right_back_desired_CR0032_temp									: WORD;(*右后垂直伸*)
	right_front_desired_temp: WORD;
	left_back_desired_temp: WORD;
	right_back_desired_temp: WORD;

	right_side_choice_m: BOOL;
	left_side_choice_m: BOOL;
END_VAR
array_cc[0].b:=cc_0;
array_cc[1].b:=cc_1;
array_cc[2].b:=cc_2;
array_cc[3].b:=cc_3;
array_cc[4].b:=cc_4;
array_cc[5].b:=cc_5;
array_cc[6].b:=cc_6;
array_cc[7].b:=cc_7;
array_cc[8].b:=cc_8;
array_cc[9].b:=cc_9;
array_cc[10].b:=cc_10;
array_cc[11].b:=cc_11;
array_cc[12].b:=cc_12;
array_cc[13].b:=cc_13;
array_cc[14].b:=cc_14;
array_cc[15].b:=cc_15;
array_cc[16].b:=cc_16;
array_cc[17].b:=cc_17;
array_cc[18].b:=cc_18;
array_cc[19].b:=cc_19;
array_cc[20].b:=cc_20;




right_side_choice_m:=0;
left_side_choice_m:=0;

IF front_right_Lv_ex_check AND back_right_Lv_ex_check THEN right_side_choice_m:=1; END_IF
IF front_left_Lv_ex_check AND back_left_Lv_ex_check THEN left_side_choice_m:=1; END_IF


IF front_left_Lv_ex_check AND back_left_Lv_ex_check AND  front_right_Lv_ex_check AND back_right_Lv_ex_check THEN
left_side_choice_m:=0; right_side_choice_m:=0;
END_IF



IF right_side_choice_m THEN
test_result:=1;
fl_A1(in:=left_front_desired,n:=4,P:=array_cc[fl_fac_r_nr2+10].b,out=>left_front_desired_CR0032);
fr_A1(in:=right_front_desired,n:=4,P:=array_cc[fr_fac_r_nr2+10].b,out=>right_front_desired_CR0032);
rl_A1(in:=left_back_desired,n:=4,P:=array_cc[rl_fac_r_nr2+10].b,out=>left_back_desired_CR0032);
rr_A1(in:=right_back_desired,n:=4,P:=array_cc[rr_fac_r_nr2+10].b,out=>right_back_desired_CR0032);
ELSIF left_side_choice_m THEN
test_result:=2;
fl_A1(in:=left_front_desired,n:=4,P:=array_cc[fl_fac_l_nr2+10].b,out=>left_front_desired_CR0032);
fr_A1(in:=right_front_desired,n:=4,P:=array_cc[fr_fac_l_nr2+10].b,out=>right_front_desired_CR0032);
rl_A1(in:=left_back_desired,n:=4,P:=array_cc[rl_fac_l_nr2+10].b,out=>left_back_desired_CR0032);
rr_A1(in:=right_back_desired,n:=4,P:=array_cc[rr_fac_l_nr2+10].b,out=>right_back_desired_CR0032);
ELSE
test_result:=3;
fl_A1(in:=left_front_desired,n:=4,P:=array_cc[fl_fac_nr2+10].b,out=>left_front_desired_CR0032);
fr_A1(in:=right_front_desired,n:=4,P:=array_cc[fr_fac_nr2+10].b,out=>right_front_desired_CR0032);
rl_A1(in:=left_back_desired,n:=4,P:=array_cc[rl_fac_nr2+10].b,out=>left_back_desired_CR0032);
rr_A1(in:=right_back_desired,n:=4,P:=array_cc[rr_fac_nr2+10].b,out=>right_back_desired_CR0032);
END_IF
END_PROGRAM

(* POU TRIGER_Regulation/case_curve, ST *)
PROGRAM case_curve
VAR

	right_temp: BOOL;
	test_result: INT;
	left_temp: BOOL;


	array_cc: ARRAY[0..20]OF cc_point;
	cc_0:ARRAY[0..10] OF POINT       :=(X:=0,Y:=0),(X:=1,Y:=100),  (X:=500,Y:=200), (X:=1000,Y:=220), 7((X:=1000,Y:=520));
	cc_1:ARRAY[0..10] OF POINT       :=(X:=0,Y:=0),(X:=1,Y:=100),  (X:=500,Y:=220), (X:=1000,Y:=240), 7((X:=1000,Y:=520));
	cc_2:ARRAY[0..10] OF POINT       :=(X:=0,Y:=0),(X:=1,Y:=100),  (X:=500,Y:=240), (X:=1000,Y:=260), 7((X:=1000,Y:=520));
	cc_3:ARRAY[0..10] OF POINT       :=(X:=0,Y:=0),(X:=1,Y:=120),  (X:=500,Y:=260), (X:=1000,Y:=300), 7((X:=1000,Y:=520));
	cc_4:ARRAY[0..10] OF POINT       :=(X:=0,Y:=0),(X:=1,Y:=140),  (X:=500,Y:=280), (X:=1000,Y:=320), 7((X:=1000,Y:=520));
	cc_5:ARRAY[0..10] OF POINT       :=(X:=0,Y:=0),(X:=1,Y:=160),  (X:=500,Y:=300), (X:=1000,Y:=340), 7((X:=1000,Y:=520));
	cc_6:ARRAY[0..10] OF POINT       :=(X:=0,Y:=0),(X:=1,Y:=180),  (X:=500,Y:=320), (X:=1000,Y:=360), 7((X:=1000,Y:=520));
	cc_7:ARRAY[0..10] OF POINT       :=(X:=0,Y:=0),(X:=1,Y:=200),  (X:=500,Y:=360), (X:=1000,Y:=400), 7((X:=1000,Y:=520));
	cc_8:ARRAY[0..10] OF POINT       :=(X:=0,Y:=0),(X:=1,Y:=220),  (X:=500,Y:=400), (X:=1000,Y:=440), 7((X:=1000,Y:=520));
	cc_9:ARRAY[0..10] OF POINT       :=(X:=0,Y:=0),(X:=1,Y:=240),  (X:=500,Y:=460), (X:=1000,Y:=480), 7((X:=1000,Y:=520));
	cc_10:ARRAY[0..10] OF POINT       :=(X:=0,Y:=0),(X:=1,Y:=260),  (X:=500,Y:=480), (X:=1000,Y:=520), 7((X:=1000,Y:=520));(*常规启动电流，对应常规支腿速度*)
	cc_11:ARRAY[0..10] OF POINT       :=(X:=0,Y:=0),(X:=1,Y:=280),  (X:=500,Y:=480), (X:=1000,Y:=520), 7((X:=1000,Y:=520));
	cc_12:ARRAY[0..10] OF POINT       :=(X:=0,Y:=0),(X:=1,Y:=280),  (X:=500,Y:=500), (X:=1000,Y:=540), 7((X:=1000,Y:=520));
	cc_13:ARRAY[0..10] OF POINT       :=(X:=0,Y:=0),(X:=1,Y:=300),  (X:=500,Y:=500), (X:=1000,Y:=540), 7((X:=1000,Y:=520));
	cc_14:ARRAY[0..10] OF POINT       :=(X:=0,Y:=0),(X:=1,Y:=300),  (X:=500,Y:=520), (X:=1000,Y:=560), 7((X:=1000,Y:=520));
	cc_15:ARRAY[0..10] OF POINT       :=(X:=0,Y:=0),(X:=1,Y:=320),  (X:=500,Y:=520), (X:=1000,Y:=560), 7((X:=1000,Y:=520));
	cc_16:ARRAY[0..10] OF POINT       :=(X:=0,Y:=0),(X:=1,Y:=320),  (X:=500,Y:=540), (X:=1000,Y:=580), 7((X:=1000,Y:=520));
	cc_17:ARRAY[0..10] OF POINT       :=(X:=0,Y:=0),(X:=1,Y:=340),  (X:=500,Y:=540), (X:=1000,Y:=580), 7((X:=1000,Y:=520));
	cc_18:ARRAY[0..10] OF POINT       :=(X:=0,Y:=0),(X:=1,Y:=360),  (X:=500,Y:=540), (X:=1000,Y:=580), 7((X:=1000,Y:=520));
	cc_19:ARRAY[0..10] OF POINT       :=(X:=0,Y:=0),(X:=1,Y:=360),  (X:=500,Y:=560), (X:=1000,Y:=600), 7((X:=1000,Y:=520));
	cc_20:ARRAY[0..10] OF POINT       :=(X:=0,Y:=0),(X:=1,Y:=400),  (X:=500,Y:=600), (X:=1000,Y:=700), 7((X:=1000,Y:=520));
	fl_A1: CHARCURVE;
	fr_A1: CHARCURVE;
	rl_A1: CHARCURVE;
	rr_A1: CHARCURVE;
	left_front_desired_temp: WORD;



	_temp										: WORD;(*左前垂直伸*)
	right_front_desired_CR0032_temp								: WORD;(*右前垂直伸*)
	left_back_desired_CR0032_temp										: WORD;(*左后垂直伸*)
	right_back_desired_CR0032_temp									: WORD;(*右后垂直伸*)
	right_front_desired_temp: WORD;
	left_back_desired_temp: WORD;
	right_back_desired_temp: WORD;

	right_side_choice_m: BOOL;
	left_side_choice_m: BOOL;
END_VAR
array_cc[0].b:=cc_0;
array_cc[1].b:=cc_1;
array_cc[2].b:=cc_2;
array_cc[3].b:=cc_3;
array_cc[4].b:=cc_4;
array_cc[5].b:=cc_5;
array_cc[6].b:=cc_6;
array_cc[7].b:=cc_7;
array_cc[8].b:=cc_8;
array_cc[9].b:=cc_9;
array_cc[10].b:=cc_10;
array_cc[11].b:=cc_11;
array_cc[12].b:=cc_12;
array_cc[13].b:=cc_13;
array_cc[14].b:=cc_14;
array_cc[15].b:=cc_15;
array_cc[16].b:=cc_16;
array_cc[17].b:=cc_17;
array_cc[18].b:=cc_18;
array_cc[19].b:=cc_19;
array_cc[20].b:=cc_20;




right_side_choice_m:=0;
left_side_choice_m:=0;

IF front_right_Lv_ex_check AND back_right_Lv_ex_check THEN right_side_choice_m:=1; END_IF
IF front_left_Lv_ex_check AND back_left_Lv_ex_check THEN left_side_choice_m:=1; END_IF


IF front_left_Lv_ex_check AND back_left_Lv_ex_check AND  front_right_Lv_ex_check AND back_right_Lv_ex_check THEN
left_side_choice_m:=0; right_side_choice_m:=0;
END_IF



IF right_side_choice_m THEN
test_result:=1;
fl_A1(in:=left_front_desired,n:=4,P:=array_cc[fl_fac_r_nr+10].b,out=>left_front_desired_CR0032);
fr_A1(in:=right_front_desired,n:=4,P:=array_cc[fr_fac_r_nr+10].b,out=>right_front_desired_CR0032);
rl_A1(in:=left_back_desired,n:=4,P:=array_cc[rl_fac_r_nr+10].b,out=>left_back_desired_CR0032);
rr_A1(in:=right_back_desired,n:=4,P:=array_cc[rr_fac_r_nr+10].b,out=>right_back_desired_CR0032);
ELSIF left_side_choice_m THEN
test_result:=2;
fl_A1(in:=left_front_desired,n:=4,P:=array_cc[fl_fac_l_nr+10].b,out=>left_front_desired_CR0032);
fr_A1(in:=right_front_desired,n:=4,P:=array_cc[fr_fac_l_nr+10].b,out=>right_front_desired_CR0032);
rl_A1(in:=left_back_desired,n:=4,P:=array_cc[rl_fac_l_nr+10].b,out=>left_back_desired_CR0032);
rr_A1(in:=right_back_desired,n:=4,P:=array_cc[rr_fac_l_nr+10].b,out=>right_back_desired_CR0032);
ELSE
test_result:=3;
fl_A1(in:=left_front_desired,n:=4,P:=array_cc[fl_fac_nr+10].b,out=>left_front_desired_CR0032);
fr_A1(in:=right_front_desired,n:=4,P:=array_cc[fr_fac_nr+10].b,out=>right_front_desired_CR0032);
rl_A1(in:=left_back_desired,n:=4,P:=array_cc[rl_fac_nr+10].b,out=>left_back_desired_CR0032);
rr_A1(in:=right_back_desired,n:=4,P:=array_cc[rr_fac_nr+10].b,out=>right_back_desired_CR0032);
END_IF
END_PROGRAM

(* POU TRIGER_Regulation/analog_in_out_cylinder, ST *)
PROGRAM analog_in_out_cylinder
VAR

END_VAR
tx_id060[0]:=INT_TO_BYTE(fl_fac_nr+50);
tx_id060[1]:=INT_TO_BYTE(fl_fac_l_nr+50);
tx_id060[2]:=INT_TO_BYTE(fl_fac_r_nr+50);
tx_id060[3]:=INT_TO_BYTE(fr_fac_nr+50);
tx_id060[4]:=INT_TO_BYTE(fr_fac_l_nr+50);
tx_id060[5]:=INT_TO_BYTE(fr_fac_r_nr+50);
tx_id060[6]:=INT_TO_BYTE(rl_fac_nr+50);
tx_id060[7]:=INT_TO_BYTE(rl_fac_l_nr+50);
tx_id061[0]:=INT_TO_BYTE(rl_fac_r_nr+50);
tx_id061[1]:=INT_TO_BYTE(rr_fac_nr+50);
tx_id061[2]:=INT_TO_BYTE(rr_fac_l_nr+50);
tx_id061[3]:=INT_TO_BYTE(rr_fac_r_nr+50);
END_PROGRAM

(* POU TRIGER_Regulation/analog_in_out_cylinder2, ST *)
PROGRAM analog_in_out_cylinder2
VAR

END_VAR
tx_id060[0]:=INT_TO_BYTE(fl_fac_nr2+50);
tx_id060[1]:=INT_TO_BYTE(fl_fac_l_nr2+50);
tx_id060[2]:=INT_TO_BYTE(fl_fac_r_nr2+50);
tx_id060[3]:=INT_TO_BYTE(fr_fac_nr2+50);
tx_id060[4]:=INT_TO_BYTE(fr_fac_l_nr2+50);
tx_id060[5]:=INT_TO_BYTE(fr_fac_r_nr2+50);
tx_id060[6]:=INT_TO_BYTE(rl_fac_nr2+50);
tx_id060[7]:=INT_TO_BYTE(rl_fac_l_nr2+50);
tx_id061[0]:=INT_TO_BYTE(rl_fac_r_nr2+50);
tx_id061[1]:=INT_TO_BYTE(rr_fac_nr2+50);
tx_id061[2]:=INT_TO_BYTE(rr_fac_l_nr2+50);
tx_id061[3]:=INT_TO_BYTE(rr_fac_r_nr2+50);
END_PROGRAM

(* POU TRIGER_LEVEL/VEHICLE/levelling2_remote2, ST *)
PROGRAM levelling2_remote2
VAR

END_VAR
level_extend_triger_left		:=	level_extend_triger_left1;
level_extend_triger_right		:=	level_extend_triger_right1;
auto_extend_triger_left		:=	auto_extend_triger_left1;
auto_extend_triger_right		:=	auto_extend_triger_right1;
auto_drawback_triger_left	:=	auto_drawback_triger_left1;
auto_drawback_triger_right	:=	auto_drawback_triger_right1;
END_PROGRAM

(* POU TRIGER_LEVEL/VEHICLE/levelling2_remote, ST *)
PROGRAM levelling2_remote
VAR
(***！！！！！！！！！！！！！！！！！！！说明！！！ 使用前请完整阅读！！！！！！！！！！！！！！！***)

(***！！！1、子程序levelling2_remote 适用于配置支腿遥控盒的车型***)

(***！！！2、对支腿操作的操作输入IO，屏蔽映射端口***)

(***！！！3、子程序levelling2_remote 需在levelling后调用 ***)

(***！！！4、remote_deal1中报警文字变量需根据车型进行修改 ***)




(***remote_pcb_in***)
	leg_choose												: BOOL;(*支腿选择*)

(***remote_pcb_out***)
	leg_choose_sign											:  BOOL;(*支腿选择*)
	lf_triger_lv_check_sign2		(*AT %QX32.10*)			:  BOOL;(*左前水平支腿伸到位信号*)
	lr_triger_lv_check_sign2		(*AT %QX32.11*)			:  BOOL;(*左后水平支腿伸到位信号*)
	rf_triger_lv_check_sign2		(*AT %QX0.14	*)			:  BOOL;(*右前水平支腿伸到位信号*)
	rr_triger_lv_check_sign2		(*AT %QX0.15	*)			:  BOOL;(*右后水平支腿伸到位信号*)
	lamp_light													:  BOOL;(*按键时照明指示*)


	CAN_REMOTE_T1	: CAN1_TRANSMIT;
	CAN_REMOTE_R1	: CAN1_RECEIVE;
	DATA_R1				: ARRAY [0..7] OF BYTE;
	DATA_T1				: ARRAY [0..7] OF BYTE;

	UNPACK1				:UNPACK;

	leg_remote_init_1	: BOOL:=1;
	leg_choose_r1		: R_TRIG;
	leaarrrrr	: R_TRIG;

	leg_choose_int		: INT:=1;

	lamp_light_t			:TON;
	lamp_light_m			:BOOL;



	aa: BOOL;
	bb: BOOL;
	ab: BOOL;
END_VAR
leg_choose							:=0;
level_extend_triger_left				:=0;
level_extend_triger_right				:=0;
auto_extend_triger_left				:=0;
auto_drawback_triger_left			:=0;
leg_choose_sign						:=0;
rf_triger_lv_check_sign2				:=0;
rr_triger_lv_check_sign2				:=0;
lf_triger_lv_check_sign2				:=0;
lr_triger_lv_check_sign2				:=0;
remote_not_arm_to_station_alarm	:=0;
remote_manual_alarm				:=0;

remote_pcb();

IF NOT leg_remote_init_1 THEN
	remote_deal1();
END_IF

remote_pcb2();

leg_remote_init_1:=0;
END_PROGRAM
ACTION remote_deal1:
IF auto_manu_choice THEN
	IF  front_left_Lv_ex_check 		THEN lf_triger_lv_check_sign2:=1;  		END_IF
	IF  back_left_Lv_ex_check 		THEN lr_triger_lv_check_sign2:=1;		END_IF
	IF  front_right_Lv_ex_check 		THEN rf_triger_lv_check_sign2:=1;		END_IF
	IF  back_right_Lv_ex_check 		THEN rr_triger_lv_check_sign2:=1;		END_IF
END_IF



leg_choose_r1(clk:=leg_choose);
IF leg_choose_r1.Q THEN
	leg_choose_int:=leg_choose_int+1;
END_IF
IF leg_choose_int=0 THEN  leg_choose_int:=1; END_IF
IF leg_choose_int>4 THEN  leg_choose_int:=1; END_IF

IF NOT auto_manu_choice THEN
	leg_choose_sign:=1;
	CASE leg_choose_int OF
		1: lf_triger_lv_check_sign2:=1;
		2: lr_triger_lv_check_sign2:=1;
		3: rf_triger_lv_check_sign2:=1;
		4: rr_triger_lv_check_sign2:=1;
	END_CASE
	IF  arm_to_station THEN
		IF lf_triger_lv_check_sign2  THEN
			IF	level_extend_triger_left		THEN	left_front_lv_ex_valve:=1;				remote_manual_alarm:=1;END_IF
			IF	level_extend_triger_right		THEN	left_front_lv_drb_valve:=1;			remote_manual_alarm:=1;END_IF
			IF	auto_extend_triger_left		THEN	left_front_desired_CR0032:=500;	remote_manual_alarm:=1;END_IF
			IF	auto_drawback_triger_left	THEN	left_front_drawback_desired:=500;	remote_manual_alarm:=1;END_IF
		END_IF
		IF lr_triger_lv_check_sign2  THEN
			IF	level_extend_triger_left		THEN	left_back_lv_ex_valve:=1;				remote_manual_alarm:=1;END_IF
			IF	level_extend_triger_right		THEN	left_back_lv_drb_valve:=1;			remote_manual_alarm:=1;END_IF
			IF	auto_extend_triger_left		THEN	left_back_desired_CR0032:=500;	remote_manual_alarm:=1;END_IF
			IF	auto_drawback_triger_left	THEN	left_back_drawback_desired:=500;	remote_manual_alarm:=1;END_IF
		END_IF
		IF rf_triger_lv_check_sign2  THEN
			IF	level_extend_triger_left		THEN	right_front_lv_drb_valve:=1;			remote_manual_alarm:=1;END_IF
			IF	level_extend_triger_right		THEN	right_front_lv_ex_valve:=1;			remote_manual_alarm:=1;END_IF
			IF	auto_extend_triger_left		THEN	right_front_desired_CR0032:=500;	remote_manual_alarm:=1;END_IF
			IF	auto_drawback_triger_left	THEN	right_front_drawback_desired:=500;	remote_manual_alarm:=1;END_IF
		END_IF
		IF rr_triger_lv_check_sign2  THEN
			IF	level_extend_triger_left		THEN	right_back_lv_drb_valve:=1;			END_IF
			IF	level_extend_triger_right		THEN	right_back_lv_ex_valve:=1;			END_IF
			IF	auto_extend_triger_left		THEN	right_back_desired_CR0032:=500;	END_IF
			IF	auto_drawback_triger_left	THEN	right_back_drawback_desired:=500;	END_IF
		END_IF
	END_IF
	IF NOT arm_to_station AND (level_extend_triger_left OR level_extend_triger_right OR auto_extend_triger_left OR auto_drawback_triger_left )THEN
			remote_not_arm_to_station_alarm:=1;
	END_IF

END_IF

(***照明指示***)
	lamp_light:=0;
	IF leg_choose OR level_extend_triger_left OR level_extend_triger_right OR auto_drawback_triger_left OR auto_extend_triger_left THEN
		lamp_light_m:=1;
	END_IF
	lamp_light_t(in:=NOT (leg_choose OR level_extend_triger_left OR level_extend_triger_right OR auto_drawback_triger_left OR auto_extend_triger_left ),pt:=t#8s );
	IF lamp_light_t.Q THEN lamp_light_m:=0;END_IF
	lamp_light:=lamp_light_m;
END_ACTION
ACTION remote_pcb:
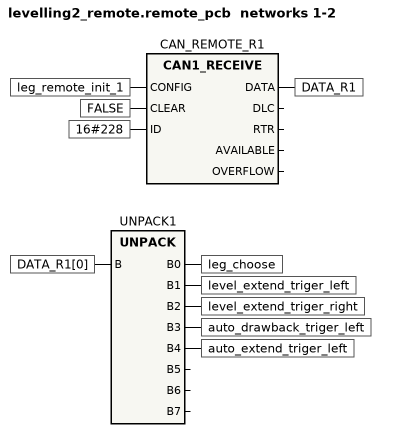
_FBD_ (* Function Block Diagram *)
NETWORK 1
	CAN_REMOTE_R1:CAN1_RECEIVE(CONFIG: leg_remote_init_1, CLEAR: FALSE, ID: 16#228) => DATA_R1
NETWORK 2
	UNPACK1:UNPACK(B: DATA_R1[0], B1 => level_extend_triger_left, B2 => level_extend_triger_right, B3 => auto_drawback_triger_left, B4 => auto_extend_triger_left) => leg_choose
_END_FBD_
(* the same logic as Structured Text *)
(* Network 1 *)
CAN_REMOTE_R1(CONFIG := leg_remote_init_1, CLEAR := FALSE, ID := 16#228);
DATA_R1 := CAN_REMOTE_R1.DATA;
(* Network 2 *)
UNPACK1(B := DATA_R1[0]);
level_extend_triger_left := UNPACK1.B1;
level_extend_triger_right := UNPACK1.B2;
auto_drawback_triger_left := UNPACK1.B3;
auto_extend_triger_left := UNPACK1.B4;
leg_choose := UNPACK1.B0;
END_ACTION
ACTION remote_pcb2:
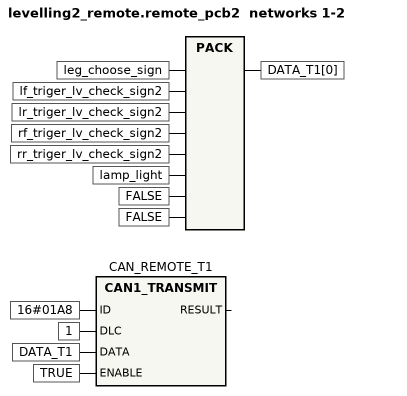
_FBD_ (* Function Block Diagram *)
NETWORK 1
	PACK(leg_choose_sign, lf_triger_lv_check_sign2, lr_triger_lv_check_sign2, rf_triger_lv_check_sign2, rr_triger_lv_check_sign2, lamp_light, FALSE, FALSE) => DATA_T1[0]
NETWORK 2
	CAN_REMOTE_T1:CAN1_TRANSMIT(ID: 16#01A8, DLC: 1, DATA: DATA_T1, ENABLE: TRUE)
_END_FBD_
(* the same logic as Structured Text *)
(* Network 1 *)
DATA_T1[0] := PACK(leg_choose_sign, lf_triger_lv_check_sign2, lr_triger_lv_check_sign2, rf_triger_lv_check_sign2, rr_triger_lv_check_sign2, lamp_light, FALSE, FALSE);
(* Network 2 *)
CAN_REMOTE_T1(ID := 16#01A8, DLC := 1, DATA := DATA_T1, ENABLE := TRUE);
END_ACTION

(* POU TRIGER_LEVEL/triger_pwm, FBD *)
PROGRAM triger_pwm
VAR
(*鉴于经常出现YT32C和YT32D的支腿单侧调平效果不理想，现增加分别对四个垂直支湍在全支撑、左单侧和右单侧模式下油缸速度进行设置修改，提高调平功能的适应范围以及可靠性***********)

	(*array_cc:ARRAY[0..2,0..10] OF cc_point:=((X:=0,Y:=0),(X:=1,Y:=260),  (X:=500,Y:=480), (X:=1000,Y:=520), 7((X:=1000,Y:=520))),((X:=0,Y:=0),(X:=1,Y:=330),  (X:=500,Y:=520), (X:=1000,Y:=600), 7((X:=1000,Y:=520))),((X:=0,Y:=0),(X:=1,Y:=160),  (X:=500,Y:=420), (X:=1000,Y:=520), 7((X:=1000,Y:=520)));

	array_cc:ARRAY[0..2] OF cc_point:=(1,(X:=0,Y:=0),(X:=1,Y:=260),  (X:=500,Y:=480), (X:=1000,Y:=520), 7((X:=1000,Y:=520))),(2,(X:=0,Y:=0),(X:=1,Y:=330),  (X:=500,Y:=520), (X:=1000,Y:=600), 7((X:=1000,Y:=520))),(3,(X:=0,Y:=0),(X:=1,Y:=160),  (X:=500,Y:=420), (X:=1000,Y:=520), 7((X:=1000,Y:=520)));

	array_cc: cc_point:=[a:=1,((X:=0,Y:=0),(X:=1,Y:=260),  (X:=500,Y:=480), (X:=1000,Y:=520), 7((X:=1000,Y:=520)))[;
*)
	cc:ARRAY[0..10] OF POINT       :=(X:=0,Y:=0),(X:=1,Y:=260),  (X:=500,Y:=480), (X:=1000,Y:=520), 7((X:=1000,Y:=520));(*常规启动电流，对应常规支腿速度*)




	left_front: OUTPUT_CURRENT_CONTROL;
	left_front_act: OUTPUT_CURRENT;

	left_front_output: WORD;
	right_front_act: OUTPUT_CURRENT;
	right_front: OUTPUT_CURRENT_CONTROL;
	right_front_output: WORD;

	left_back: OUTPUT_CURRENT_CONTROL;
	left_back_act: OUTPUT_CURRENT;
	left_back_output: WORD;

	right_back: OUTPUT_CURRENT_CONTROL;
	right_back_output: WORD;
	right_back_act: OUTPUT_CURRENT;

	right_front_drawback: OUTPUT_CURRENT_CONTROL;
	right_front_drawback_act: OUTPUT_CURRENT;

	right_front_drawback_output: WORD;
	left_back_drawback: OUTPUT_CURRENT_CONTROL;
	left_back_drawback_output: WORD;

	left_back_drawback_act: OUTPUT_CURRENT;
	right_back_drawback: OUTPUT_CURRENT_CONTROL;
	right_back_drawback_output: WORD;
	right_back_drawback_act: OUTPUT_CURRENT;

	left_front_drawback: OUTPUT_CURRENT_CONTROL;
	left_front_drawback_act: OUTPUT_CURRENT;
	left_front_drawback_output: WORD;

	A1: CHARCURVE;
	a2: WORD;
	a3: INT;

	x1: REAL;
	left_front_occ: CONTROL_OCC;
	right_back_occ: CONTROL_OCC;
	left_back_occ: CONTROL_OCC;
	right_front_occ: CONTROL_OCC;

	left_front_r_occ: CONTROL_OCC;
	right_back_r_occ: CONTROL_OCC;
	left_back_r_occ: CONTROL_OCC;
	right_front_r_occ: CONTROL_OCC;
END_VAR
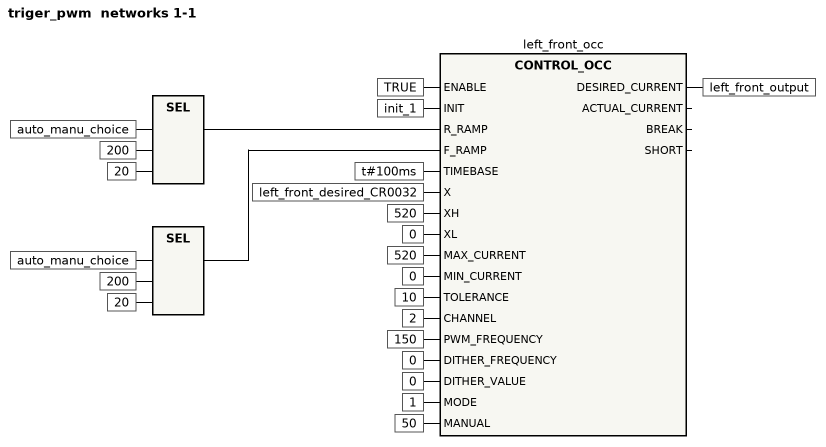
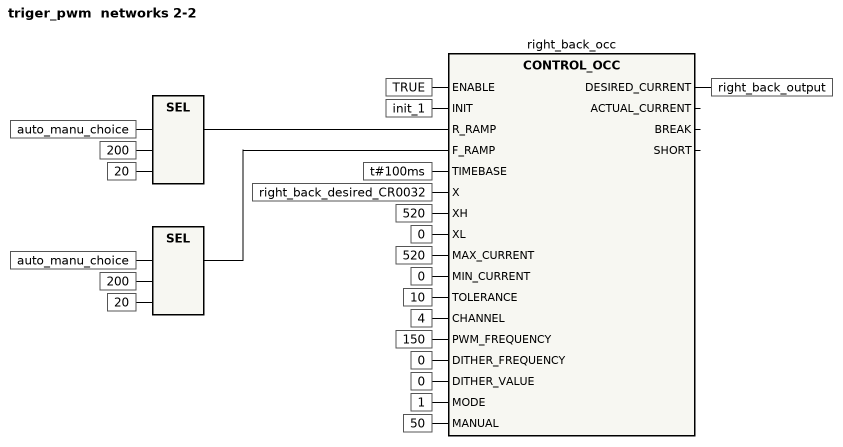
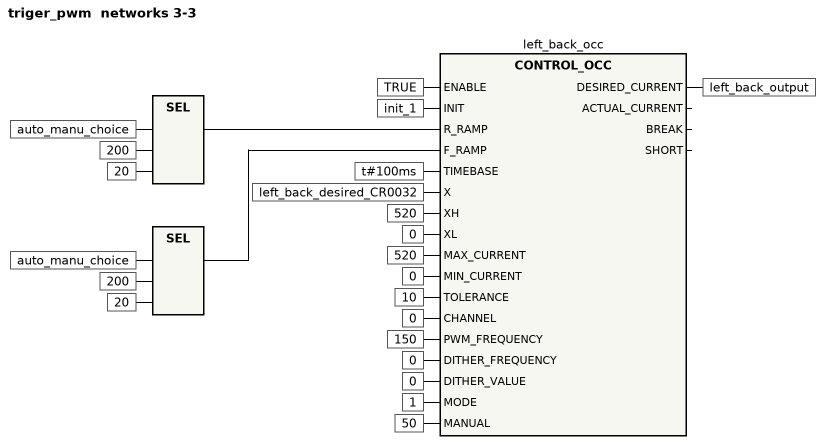
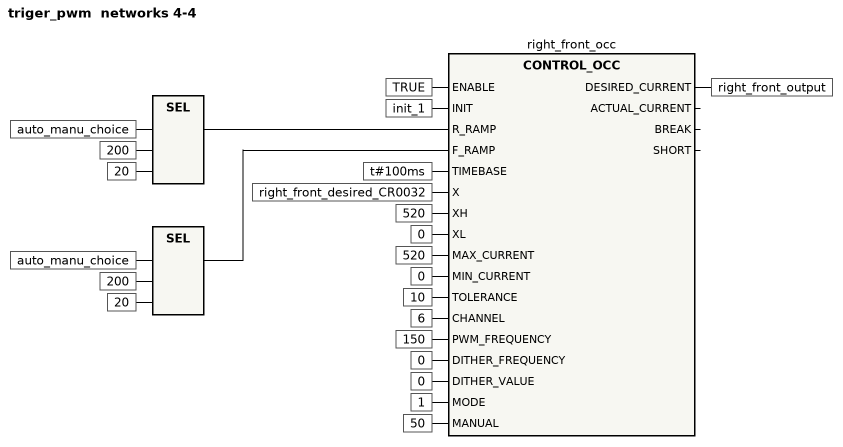
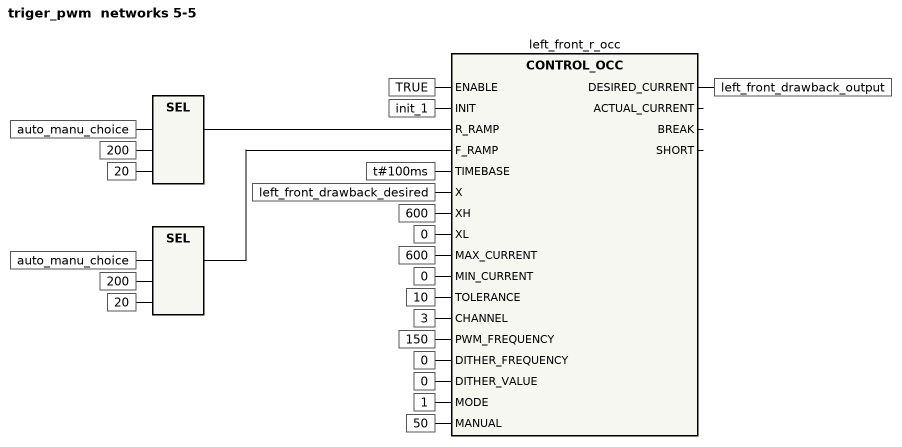
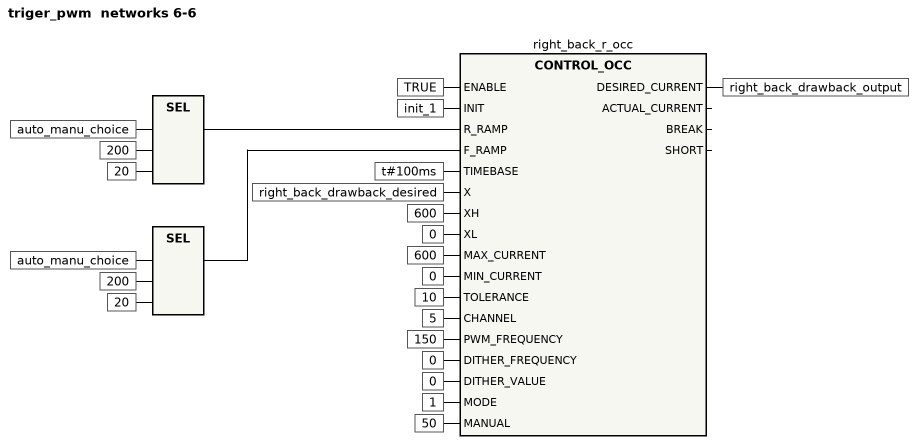
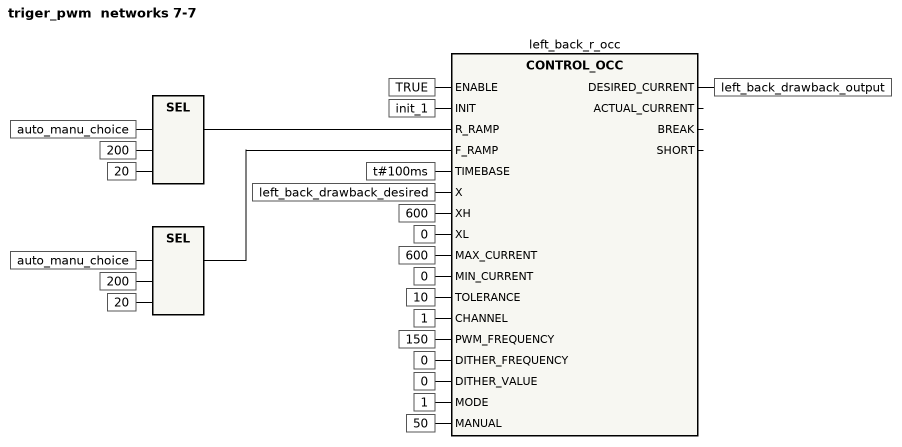
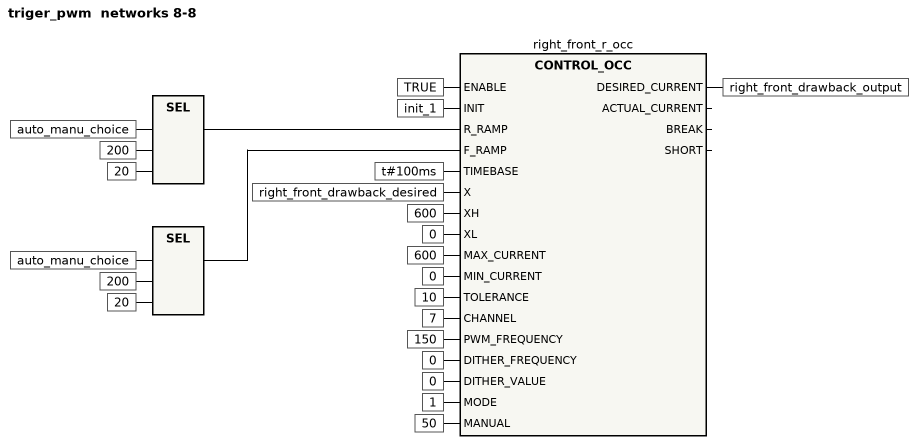
_FBD_ (* Function Block Diagram *)
NETWORK 1 (* 1、左前垂直伸速度控制段，第一个ccX处表示全支撑模式速度，第二个ccX处表示左单侧支撑模式速度，第三个ccX处表示右单侧支撑模式速度。其中，ccX代表cc、cc1或者cc2。 / 2、调试时某种模式速度不理想，在对应位置ccX重新选择，ccX具体数值参考上面的变量申明处内容。 / 3、如果已提供的三组ccX（cc、cc1和cc2）仍然无法满足调平功能需求，建议重新定义一组新的ccX，把x=1、x=500和x=1000对应的三处Y值分别增加或者减小。 / 举例说明：如果第一个cc2改成cc1，表示全支撑模式下的左前垂直油缸速度从慢档速度设置成快档速度。 *)
	left_front_occ:CONTROL_OCC(ENABLE: TRUE, INIT: init_1, R_RAMP: SEL(auto_manu_choice, 200, 20), F_RAMP: SEL(auto_manu_choice, 200, 20), TIMEBASE: t#100ms, X: left_front_desired_CR0032, XH: 520, XL: 0, MAX_CURRENT: 520, MIN_CURRENT: 0, TOLERANCE: 10, CHANNEL: 2, PWM_FREQUENCY: 150, DITHER_FREQUENCY: 0, DITHER_VALUE: 0, MODE: 1, MANUAL: 50) => left_front_output
NETWORK 2 (* 1、右后垂直伸速度控制段，第一个ccX处表示全支撑模式速度，第二个ccX处表示左单侧支撑模式速度，第三个ccX处表示右单侧支撑模式速度。其中，ccX代表cc、cc1或者cc2。 / 2、调试时某种模式速度不理想，在对应位置ccX重新选择，ccX具体数值参考上面的变量申明处内容。 / 3、如果已提供的三组ccX（cc、cc1和cc2）仍然无法满足调平功能需求，建议重新定义一组新的ccX，把x=1、x=500和x=1000对应的Y值分别增加或者减小。 / 举例说明：如果第一个cc改成cc1，表示全支撑模式下的右后垂直油缸速度从常规速度设置成快档速度。 *)
	right_back_occ:CONTROL_OCC(ENABLE: TRUE, INIT: init_1, R_RAMP: SEL(auto_manu_choice, 200, 20), F_RAMP: SEL(auto_manu_choice, 200, 20), TIMEBASE: t#100ms, X: right_back_desired_CR0032, XH: 520, XL: 0, MAX_CURRENT: 520, MIN_CURRENT: 0, TOLERANCE: 10, CHANNEL: 4, PWM_FREQUENCY: 150, DITHER_FREQUENCY: 0, DITHER_VALUE: 0, MODE: 1, MANUAL: 50) => right_back_output
NETWORK 3 (* 1、左后垂直伸速度控制段，第一个ccX处表示全支撑模式速度，第二个ccX处表示左单侧支撑模式速度，第三个ccX处表示右单侧支撑模式速度。其中，ccX代表cc、cc1或者cc2。 / 2、调试时某种模式速度不理想，在对应位置ccX重新选择，ccX具体数值参考上面的变量申明处内容。 / 3、如果已提供的三组ccX（cc、cc1和cc2）仍然无法满足调平功能需求，建议重新定义一组新的ccX，把x=1、x=500和x=1000对应的Y值分别增加或者减小。 / 举例说明：如果第一个cc2改成cc1，表示全支撑模式下的左后垂直油缸速度从慢档速度设置成快档速度。 *)
	left_back_occ:CONTROL_OCC(ENABLE: TRUE, INIT: init_1, R_RAMP: SEL(auto_manu_choice, 200, 20), F_RAMP: SEL(auto_manu_choice, 200, 20), TIMEBASE: t#100ms, X: left_back_desired_CR0032, XH: 520, XL: 0, MAX_CURRENT: 520, MIN_CURRENT: 0, TOLERANCE: 10, CHANNEL: 0, PWM_FREQUENCY: 150, DITHER_FREQUENCY: 0, DITHER_VALUE: 0, MODE: 1, MANUAL: 50) => left_back_output
NETWORK 4 (* 1、右前垂直伸速度控制段，第一个ccX处表示全支撑模式速度，第二个ccX处表示左单侧支撑模式速度，第三个ccX处表示右单侧支撑模式速度。其中，ccX代表cc、cc1或者cc2。 / 2、调试时某种模式速度不理想，在对应位置ccX重新选择，ccX具体数值参考上面的变量申明处内容。 / 3、如果已提供的三组ccX（cc、cc1和cc2）仍然无法满足调平功能需求，建议重新定义一组新的ccX，把x=1、x=500和x=1000对应的Y值分别增加或者减小。 / 举例说明：如果第一个cc改成cc1，表示全支撑模式下的右前垂直油缸速度从常规速度设置成快档速度。 *)
	right_front_occ:CONTROL_OCC(ENABLE: TRUE, INIT: init_1, R_RAMP: SEL(auto_manu_choice, 200, 20), F_RAMP: SEL(auto_manu_choice, 200, 20), TIMEBASE: t#100ms, X: right_front_desired_CR0032, XH: 520, XL: 0, MAX_CURRENT: 520, MIN_CURRENT: 0, TOLERANCE: 10, CHANNEL: 6, PWM_FREQUENCY: 150, DITHER_FREQUENCY: 0, DITHER_VALUE: 0, MODE: 1, MANUAL: 50) => right_front_output
NETWORK 5
	left_front_r_occ:CONTROL_OCC(ENABLE: TRUE, INIT: init_1, R_RAMP: SEL(auto_manu_choice, 200, 20), F_RAMP: SEL(auto_manu_choice, 200, 20), TIMEBASE: t#100ms, X: left_front_drawback_desired, XH: 600, XL: 0, MAX_CURRENT: 600, MIN_CURRENT: 0, TOLERANCE: 10, CHANNEL: 3, PWM_FREQUENCY: 150, DITHER_FREQUENCY: 0, DITHER_VALUE: 0, MODE: 1, MANUAL: 50) => left_front_drawback_output
NETWORK 6
	right_back_r_occ:CONTROL_OCC(ENABLE: TRUE, INIT: init_1, R_RAMP: SEL(auto_manu_choice, 200, 20), F_RAMP: SEL(auto_manu_choice, 200, 20), TIMEBASE: t#100ms, X: right_back_drawback_desired, XH: 600, XL: 0, MAX_CURRENT: 600, MIN_CURRENT: 0, TOLERANCE: 10, CHANNEL: 5, PWM_FREQUENCY: 150, DITHER_FREQUENCY: 0, DITHER_VALUE: 0, MODE: 1, MANUAL: 50) => right_back_drawback_output
NETWORK 7
	left_back_r_occ:CONTROL_OCC(ENABLE: TRUE, INIT: init_1, R_RAMP: SEL(auto_manu_choice, 200, 20), F_RAMP: SEL(auto_manu_choice, 200, 20), TIMEBASE: t#100ms, X: left_back_drawback_desired, XH: 600, XL: 0, MAX_CURRENT: 600, MIN_CURRENT: 0, TOLERANCE: 10, CHANNEL: 1, PWM_FREQUENCY: 150, DITHER_FREQUENCY: 0, DITHER_VALUE: 0, MODE: 1, MANUAL: 50) => left_back_drawback_output
NETWORK 8
	right_front_r_occ:CONTROL_OCC(ENABLE: TRUE, INIT: init_1, R_RAMP: SEL(auto_manu_choice, 200, 20), F_RAMP: SEL(auto_manu_choice, 200, 20), TIMEBASE: t#100ms, X: right_front_drawback_desired, XH: 600, XL: 0, MAX_CURRENT: 600, MIN_CURRENT: 0, TOLERANCE: 10, CHANNEL: 7, PWM_FREQUENCY: 150, DITHER_FREQUENCY: 0, DITHER_VALUE: 0, MODE: 1, MANUAL: 50) => right_front_drawback_output
_END_FBD_
(* the same logic as Structured Text *)
(* Network 1: 1、左前垂直伸速度控制段，第一个ccX处表示全支撑模式速度，第二个ccX处表示左单侧支撑模式速度，第三个ccX处表示右单侧支撑模式速度。其中，ccX代表cc、cc1或者cc2。 / 2、调试时某种模式速度不理想，在对应位置ccX重新选择，ccX具体数值参考上面的变量申明处内容。 / 3、如果已提供的三组ccX（cc、cc1和cc2）仍然无法满足调平功能需求，建议重新定义一组新的ccX，把x=1、x=500和x=1000对应的三处Y值分别增加或者减小。 / 举例说明：如果第一个cc2改成cc1，表示全支撑模式下的左前垂直油缸速度从慢档速度设置成快档速度。 *)
left_front_occ(ENABLE := TRUE, INIT := init_1, R_RAMP := SEL(auto_manu_choice, 200, 20), F_RAMP := SEL(auto_manu_choice, 200, 20), TIMEBASE := t#100ms, X := left_front_desired_CR0032, XH := 520, XL := 0, MAX_CURRENT := 520, MIN_CURRENT := 0, TOLERANCE := 10, CHANNEL := 2, PWM_FREQUENCY := 150, DITHER_FREQUENCY := 0, DITHER_VALUE := 0, MODE := 1, MANUAL := 50);
left_front_output := left_front_occ.DESIRED_CURRENT;
(* Network 2: 1、右后垂直伸速度控制段，第一个ccX处表示全支撑模式速度，第二个ccX处表示左单侧支撑模式速度，第三个ccX处表示右单侧支撑模式速度。其中，ccX代表cc、cc1或者cc2。 / 2、调试时某种模式速度不理想，在对应位置ccX重新选择，ccX具体数值参考上面的变量申明处内容。 / 3、如果已提供的三组ccX（cc、cc1和cc2）仍然无法满足调平功能需求，建议重新定义一组新的ccX，把x=1、x=500和x=1000对应的Y值分别增加或者减小。 / 举例说明：如果第一个cc改成cc1，表示全支撑模式下的右后垂直油缸速度从常规速度设置成快档速度。 *)
right_back_occ(ENABLE := TRUE, INIT := init_1, R_RAMP := SEL(auto_manu_choice, 200, 20), F_RAMP := SEL(auto_manu_choice, 200, 20), TIMEBASE := t#100ms, X := right_back_desired_CR0032, XH := 520, XL := 0, MAX_CURRENT := 520, MIN_CURRENT := 0, TOLERANCE := 10, CHANNEL := 4, PWM_FREQUENCY := 150, DITHER_FREQUENCY := 0, DITHER_VALUE := 0, MODE := 1, MANUAL := 50);
right_back_output := right_back_occ.DESIRED_CURRENT;
(* Network 3: 1、左后垂直伸速度控制段，第一个ccX处表示全支撑模式速度，第二个ccX处表示左单侧支撑模式速度，第三个ccX处表示右单侧支撑模式速度。其中，ccX代表cc、cc1或者cc2。 / 2、调试时某种模式速度不理想，在对应位置ccX重新选择，ccX具体数值参考上面的变量申明处内容。 / 3、如果已提供的三组ccX（cc、cc1和cc2）仍然无法满足调平功能需求，建议重新定义一组新的ccX，把x=1、x=500和x=1000对应的Y值分别增加或者减小。 / 举例说明：如果第一个cc2改成cc1，表示全支撑模式下的左后垂直油缸速度从慢档速度设置成快档速度。 *)
left_back_occ(ENABLE := TRUE, INIT := init_1, R_RAMP := SEL(auto_manu_choice, 200, 20), F_RAMP := SEL(auto_manu_choice, 200, 20), TIMEBASE := t#100ms, X := left_back_desired_CR0032, XH := 520, XL := 0, MAX_CURRENT := 520, MIN_CURRENT := 0, TOLERANCE := 10, CHANNEL := 0, PWM_FREQUENCY := 150, DITHER_FREQUENCY := 0, DITHER_VALUE := 0, MODE := 1, MANUAL := 50);
left_back_output := left_back_occ.DESIRED_CURRENT;
(* Network 4: 1、右前垂直伸速度控制段，第一个ccX处表示全支撑模式速度，第二个ccX处表示左单侧支撑模式速度，第三个ccX处表示右单侧支撑模式速度。其中，ccX代表cc、cc1或者cc2。 / 2、调试时某种模式速度不理想，在对应位置ccX重新选择，ccX具体数值参考上面的变量申明处内容。 / 3、如果已提供的三组ccX（cc、cc1和cc2）仍然无法满足调平功能需求，建议重新定义一组新的ccX，把x=1、x=500和x=1000对应的Y值分别增加或者减小。 / 举例说明：如果第一个cc改成cc1，表示全支撑模式下的右前垂直油缸速度从常规速度设置成快档速度。 *)
right_front_occ(ENABLE := TRUE, INIT := init_1, R_RAMP := SEL(auto_manu_choice, 200, 20), F_RAMP := SEL(auto_manu_choice, 200, 20), TIMEBASE := t#100ms, X := right_front_desired_CR0032, XH := 520, XL := 0, MAX_CURRENT := 520, MIN_CURRENT := 0, TOLERANCE := 10, CHANNEL := 6, PWM_FREQUENCY := 150, DITHER_FREQUENCY := 0, DITHER_VALUE := 0, MODE := 1, MANUAL := 50);
right_front_output := right_front_occ.DESIRED_CURRENT;
(* Network 5 *)
left_front_r_occ(ENABLE := TRUE, INIT := init_1, R_RAMP := SEL(auto_manu_choice, 200, 20), F_RAMP := SEL(auto_manu_choice, 200, 20), TIMEBASE := t#100ms, X := left_front_drawback_desired, XH := 600, XL := 0, MAX_CURRENT := 600, MIN_CURRENT := 0, TOLERANCE := 10, CHANNEL := 3, PWM_FREQUENCY := 150, DITHER_FREQUENCY := 0, DITHER_VALUE := 0, MODE := 1, MANUAL := 50);
left_front_drawback_output := left_front_r_occ.DESIRED_CURRENT;
(* Network 6 *)
right_back_r_occ(ENABLE := TRUE, INIT := init_1, R_RAMP := SEL(auto_manu_choice, 200, 20), F_RAMP := SEL(auto_manu_choice, 200, 20), TIMEBASE := t#100ms, X := right_back_drawback_desired, XH := 600, XL := 0, MAX_CURRENT := 600, MIN_CURRENT := 0, TOLERANCE := 10, CHANNEL := 5, PWM_FREQUENCY := 150, DITHER_FREQUENCY := 0, DITHER_VALUE := 0, MODE := 1, MANUAL := 50);
right_back_drawback_output := right_back_r_occ.DESIRED_CURRENT;
(* Network 7 *)
left_back_r_occ(ENABLE := TRUE, INIT := init_1, R_RAMP := SEL(auto_manu_choice, 200, 20), F_RAMP := SEL(auto_manu_choice, 200, 20), TIMEBASE := t#100ms, X := left_back_drawback_desired, XH := 600, XL := 0, MAX_CURRENT := 600, MIN_CURRENT := 0, TOLERANCE := 10, CHANNEL := 1, PWM_FREQUENCY := 150, DITHER_FREQUENCY := 0, DITHER_VALUE := 0, MODE := 1, MANUAL := 50);
left_back_drawback_output := left_back_r_occ.DESIRED_CURRENT;
(* Network 8 *)
right_front_r_occ(ENABLE := TRUE, INIT := init_1, R_RAMP := SEL(auto_manu_choice, 200, 20), F_RAMP := SEL(auto_manu_choice, 200, 20), TIMEBASE := t#100ms, X := right_front_drawback_desired, XH := 600, XL := 0, MAX_CURRENT := 600, MIN_CURRENT := 0, TOLERANCE := 10, CHANNEL := 7, PWM_FREQUENCY := 150, DITHER_FREQUENCY := 0, DITHER_VALUE := 0, MODE := 1, MANUAL := 50);
right_front_drawback_output := right_front_r_occ.DESIRED_CURRENT;
END_PROGRAM

(* POU UNDER_DEALING/DOWN_PART_DEAL, ST *)
PROGRAM DOWN_PART_DEAL
VAR
	alarmer_horn1	:BOOL;
	alarmer_horn_r	:R_TRIG;
	alarmer_horn_m	:BOOL;
	alarmer_horn_t	:TON;

	beep_set_1		: BLINK;
	beep_set_2		: BLINK;
	beep_set_2_M	: BOOL;
	T_beep_set_2	: TON;
	manual_l_r_trig	:R_TRIG;

	R_TRIG1: R_TRIG;

	up_valve_ctl_t: TON;
	up_valve_ctl_m: BOOL;
	right_lv_ex_over: BOOL;
	left_lv_ex_over: BOOL;

	ton_stop1: TON;
	ton_stop2: TON;
	stop_m: BOOL;

	xx: BOOL;

	beep_set_3_M	: BOOL;
	T_beep_set_3	: TON;
	arm_to_station_r			:R_TRIG;

	auto_manu_choice_r		: R_TRIG;
	mv_alarm10009_m		: BOOL;
	mv_alarm10009_t		: TON;

	leveled_r					: R_TRIG;
	mv_alarm10010_m		: BOOL;
	mv_alarm10010_t		: TON;

	water_pump_ctl_r			: R_TRIG;
	mv_alarm10015_m		: BOOL;
	mv_alarm10015_t		: TON;


	PTO_T1					: TON;
	PTO_M1					: BOOL;
	PTO_T2					: TON;
	PTO_M2					: BOOL;
	PTO_T3					: TON;
	PTO_M3					: BOOL;

END_VAR
down_deal();

CASE vehicle_styel OF
10011:
	add_100();
10012:
	add_10012();
10013:
	add_100();
10014:
	add_100();
ELSE
	add_100();
END_CASE
END_PROGRAM
ACTION add_100:
;
END_ACTION
ACTION add_10012:
(******************************PTO**********************************)
PTO_T1(IN:=(speed_sign>200), PT:=T#3S);
IF PTO_T1.Q THEN PTO_M1:=1; END_IF
PTO_T2(IN:=(PTO_M1), PT:=T#1.8S);
IF PTO_T2.Q THEN PTO_M2:=1; END_IF
PTO_T3(IN:=(PTO_M2), PT:=T#3S);
IF PTO_T3.Q THEN PTO_M3:=1; END_IF

IF PTO_M1 AND NOT PTO_M2  THEN enginer_acc_ctl:=1; END_IF
IF speed_sign=0 OR(PTO_M1 =0 AND PTO_M2 =0 AND PTO_M3 =0)OR (PTO_M1 AND(PTO_M2 AND NOT PTO_M3)) THEN enginer_acc_ctl:=0; END_IF
IF speed_sign=0 THEN PTO_M1:=0; PTO_M2:=0; PTO_M3:=0; PTO_T1(in:=0); PTO_T2(in:=0); PTO_T3(in:=0);END_IF
END_ACTION
ACTION down_deal:
(*************************************************操作输出*************************************************)
(******************************启动熄火*********************************)
	IF (engine_stop AND NOT stage_engine_startup AND NOT tt_engine_startup)OR(stage_engine_stop AND NOT tt_engine_startup AND NOT engine_run)
		OR (tt_engine_stop AND NOT engine_run AND NOT stage_engine_startup) THEN
		enginer_stop_ctl:=1;
		mv_alarm10002:=1;
	ELSE
		enginer_stop_ctl:=0;
	END_IF
	ton_stop1(in:=(engine_stop AND NOT stage_engine_startup AND NOT tt_engine_startup)OR(stage_engine_stop AND NOT tt_engine_startup AND NOT engine_run)
		OR (tt_engine_stop AND NOT engine_run AND NOT stage_engine_startup),Pt:=t#0.2s);
	IF ton_stop1.Q THEN stop_m:=1; END_IF
	ton_stop2(in:=stop_m,pt:=t#5s);
	IF ton_stop2.Q THEN stop_m:=0; END_IF
	IF stop_m THEN enginer_stop_ctl:=1; END_IF

	IF (engine_run AND NOT stage_engine_stop AND NOT tt_engine_stop)OR(stage_engine_startup AND NOT engine_stop AND NOT tt_engine_stop)
		OR (tt_engine_startup AND NOT stage_engine_stop AND NOT engine_stop) THEN
		enginer_run_ctl:=1; stop_m:=0;
		mv_alarm10001:=1;
	ELSE
		enginer_run_ctl:=0;
	END_IF
	IF enginer_run_ctl THEN enginer_stop_ctl:=0; END_IF
	IF enginer_stop_ctl THEN enginer_run_ctl:=0; END_IF

(**********************************应急泵************************************)
IF sudden_pump_button OR tt_emergency_pump  OR standby_pump_check THEN
	standby_oil_pump:=1;
ELSE
	standby_oil_pump:=0;
END_IF

(***************************消防泵启动停止*****************************)
R_TRIG1(CLK:= water_pump_run_sb OR  stage_water_pump_open OR tt_water_pump_open);
 IF R_TRIG1.Q THEN water_pump_ctl:=NOT water_pump_ctl;	END_IF

(******************************加减速度**********************************)
IF water_pump_ctl AND cruise_sign_set AND  speed_sign>135   THEN
	IF accelerate_sb OR stage_engine_acc OR tt_engine_acc AND NOT enginer_dec_ctl AND NOT(	(error1 OR	error2)AND NOT water_alarm_c  )THEN
		enginer_acc_ctl:=1;
	ELSE
		enginer_acc_ctl:=0;
	END_IF
	IF (stage_engine_dec OR decelerate_sb OR tt_engine_dec  AND NOT enginer_acc_ctl) OR (error2 AND NOT water_alarm_c)  THEN
		enginer_dec_ctl:=1;
	ELSE
		enginer_dec_ctl:=0;
	END_IF
END_IF

(***************************上下车阀门控制*****************************)
up_valve_ctl_t(in:=up_valve_ctl_m,pt:=t#1s);
IF up_valve_ctl_t.Q  AND speed_m<200 THEN
	up_valve_ctl		:=0;
END_IF
down_valve_ctl		:=0;
(*下车阀控制*)
IF((down_force AND arm_to_station AND NOT up_valve_ctl) OR (NOT  auto_manu_choice AND arm_to_station)OR extend_left_lv_triger_act OR extend_right_lv_triger_act OR (extend_do AND NOT (extend_step=7))OR(withdraw_do AND NOT (withdraw_step=10))  )AND NOT up_valve_ctl
	THEN
		down_valve_ctl:=1;
		up_valve_ctl_m:=0;
END_IF
(*上车阀控制*)
IF((((tt_forcexx) OR (NOT up_down_switch AND  tt_foot_switch) OR (up_down_switch AND  stage_foot_switch)) AND leveled))AND NOT down_valve_ctl
	THEN
		up_valve_ctl:=1;
		down_valve_ctl:=0;
		up_valve_ctl_m:=0;
	ELSE
		up_valve_ctl_m:=1;
END_IF
(*倾角传感器故障*)
	IF angle_x>angle_danger02+200 OR angle_x<angle_danger01-200 THEN
(*
		down_valve_ctl:=0;
		up_valve_ctl:=0;
*)	
		alarmer_horn1:=beep_set_1.OUT;
		mv_alarm10003:=1;
	END_IF



(***********************************************报警及指示等***********************************************)
alarmer_horn:=0;
alarmer_horn1:=0;

beep_set_1(ENABLE:=TRUE , TIMELOW:=t#900ms , TIMEHIGH:=t#500ms);
beep_signal:=beep_set_1.OUT;

triger_left_ground_for:=0;
IF leveled THEN
	IF NOT front_left_urt_ex_check THEN
		triger_left_ground_for:=triger_left_ground_for+1;
	END_IF
	IF NOT front_right_urt_ex_check THEN
		triger_left_ground_for:=triger_left_ground_for+1;
	END_IF
	IF NOT back_left_urt_ex_check THEN
		triger_left_ground_for:=triger_left_ground_for+1;
	END_IF
	IF NOT back_right_urt_ex_check THEN
		triger_left_ground_for:=triger_left_ground_for+1;
	END_IF
ELSE
	triger_left_ground_for:=0;
END_IF

(****************************报警**************************)
(***手动调平调平报警***)
manual_l_r_trig(CLK:=leveled);
IF NOT auto_manu_choice THEN
	IF manual_l_r_trig.Q THEN
		beep_set_2_M:=1;
	END_IF
	IF beep_set_2_M THEN
		T_beep_set_2(IN:=1,PT:=T#1S);
		beep_set_2(ENABLE:=TRUE , TIMELOW:=t#900ms , TIMEHIGH:=t#500ms);
		alarmer_horn1:=beep_set_2.OUT;
	END_IF
	IF T_beep_set_2.Q THEN
		T_beep_set_2(IN:=0);
		beep_set_2_M:=0;
	END_IF
END_IF

(***支腿离地报警***)
IF triger_left_ground_for=1  THEN
	alarmer_horn1:=beep_set_1.OUT;
END_IF

(***强制报警***)
IF down_force AND down_valve_ctl THEN
	alarmer_horn1:=beep_set_1.OUT;
	mv_alarm10004:=1;
END_IF

(***转台关联报警***)
IF NOT leveled AND((NOT up_down_switch AND  tt_foot_switch) OR (up_down_switch AND  stage_foot_switch)) THEN
	alarmer_horn1:=beep_set_1.OUT;
	mv_alarm10005:=1;
END_IF

(***臂架到位3声报警***)
arm_to_station_r(CLK:=arm_to_station);
IF arm_to_station_r.Q  THEN
	beep_set_3_M:=1;
END_IF
IF beep_set_3_M THEN
	mv_alarm10008:=1;
	T_beep_set_3(IN:=1,PT:=T#1.8S);
	alarmer_horn1:=beep_set_1.OUT;
END_IF
IF T_beep_set_3.Q THEN
	T_beep_set_3(IN:=0);
	beep_set_3_M:=0;
END_IF


(***水泡压力超压报警***)
IF error1 THEN 	alarmer_horn1:=beep_set_1.OUT; 		END_IF
IF error2 THEN 	alarmer_horn1:=1; 						END_IF

(*支腿遥控器报警*)
IF remote_manual_alarm OR remote_not_arm_to_station_alarm THEN
	alarmer_horn1:=beep_set_1.OUT;
END_IF

(***动作及虚腿报警***)
IF angle_x>angle_danger02 OR angle_x<angle_danger01 OR extend_left_lv_triger_act OR extend_right_lv_triger_act OR  extend_do OR withdraw_do OR over_level_sign OR triger_left_ground_for>=2 THEN
	alarmer_horn1:=1;
END_IF

(***通信故障报警***)
IF mv_alarm10007 THEN
	alarmer_horn1:=beep_set_1.OUT;
END_IF

(***报警声维持***)
alarmer_horn_r(clk:=alarmer_horn1);
IF alarmer_horn_r.Q THEN alarmer_horn_m:=1; END_IF
alarmer_horn_t(in:=alarmer_horn_m,pt:=t#0.4s);
IF alarmer_horn_t.Q THEN alarmer_horn_m:=0; END_IF
IF NOT frequ_set THEN
	alarmer_horn:=alarmer_horn1 OR alarmer_horn_m;
END_IF

(****************************指示**************************)
(***水平到位指示***)
IF(front_left_Lv_ex_check)			THEN 	left_f_lv_ex_over:=1;			ELSE	 	left_f_lv_ex_over:=0;		END_IF
IF(back_left_Lv_ex_check)			THEN 	left_b_lv_ex_over:=1;			ELSE	 	left_b_lv_ex_over:=0;		END_IF
IF(front_right_Lv_ex_check)			THEN 	right_f_lv_ex_over:=1;			ELSE	 	right_f_lv_ex_over:=0;		END_IF
IF(back_right_Lv_ex_check)			THEN 	right_b_lv_ex_over:=1;		ELSE	 	right_b_lv_ex_over:=0;	END_IF

(***手动操作下车指示***)
auto_manu_choice_r(CLK:=NOT auto_manu_choice);
IF auto_manu_choice_r.Q THEN mv_alarm10009_m:=1;	END_IF
IF mv_alarm10009_m THEN
	mv_alarm10009:=1;
	mv_alarm10009_t(IN:=1,PT:=T#1.8S);
END_IF
IF mv_alarm10009_t.Q THEN
	mv_alarm10009_t(in:=0);
	mv_alarm10009_m:=0;
END_IF

(***下车调平指示***)
leveled_r(CLK:=leveled);
IF leveled_r.Q THEN mv_alarm10010_m:=1;	END_IF
IF mv_alarm10010_m THEN
	mv_alarm10010:=1;
	mv_alarm10010_t(IN:=1,PT:=T#1.8S);
END_IF
IF mv_alarm10010_t.Q THEN
	mv_alarm10010_t(in:=0);
	mv_alarm10010_m:=0;
END_IF

(***水泵启动指示***)
water_pump_ctl_r(CLK:=water_pump_ctl);
IF water_pump_ctl_r.Q THEN mv_alarm10015_m:=1;	END_IF
IF mv_alarm10015_m THEN
	mv_alarm10015:=1;
	mv_alarm10015_t(IN:=1,PT:=T#1.8S);
END_IF
IF mv_alarm10015_t.Q THEN
	mv_alarm10015_t(in:=0);
	mv_alarm10015_m:=0;
END_IF

(***坡度超限指示***)
IF ABS(angle_x-angle_x_offset)>400 OR ABS(angle_y-angle_y_offset)>400 OR angle_x>angle_danger02 OR angle_x<angle_danger01 THEN
	over_level_sign:=beep_set_1.OUT;
	alarmer_horn1:=beep_set_1.OUT;
	IF NOT mv_alarm10003  THEN mv_alarm10006:=1; END_IF
ELSE
	over_level_sign:=0;
END_IF

(***上下车阀工作指示***)
down_work_sign	:=down_valve_ctl;
up_work_sign		:=up_valve_ctl;

(***支腿未全缩指示灯***)
IF NOT( front_left_Lv_drb_check AND front_right_Lv_drb_check  AND back_left_Lv_drb_check AND back_right_Lv_drb_check)THEN
	triger_flash:=1;
	triger_no_drawback_sign:=1;
ELSE
	triger_flash:=0;
	triger_no_drawback_sign:=0;
END_IF

(***调平后支腿离地指示***)
IF triger_left_ground_for>=1 THEN
	triger_left_grd_sign:=1;
ELSE
	triger_left_grd_sign:=0;
END_IF

(***支腿调平指示灯***)
leveled_sign:=leveled;

(***水泵工作指示***)
IF water_pump_ctl THEN
	water_pump_ctl_sign	:=1;
ELSE
	water_pump_ctl_sign	:=0;
END_IF
END_ACTION

(* POU COM_ERROR, ST *)
PROGRAM COM_ERROR
VAR
	ton_turn_p:TON;
	ton_turn_n:TON;

	ton_stage_p:TON;
	ton_stage_n:TON;
END_VAR
	ton_turn_p(in:=tt_turn_com,pt:=t#3s);
	ton_turn_n(in:=NOT tt_turn_com,pt:=t#3s);

	ton_stage_p(in:=stage_com,pt:=t#3s);
	ton_stage_n(in:=NOT stage_com,pt:=t#3s);

	IF ton_turn_p.Q OR ton_turn_n.Q OR ton_stage_p.Q OR ton_stage_n.Q THEN
		up_valve_ctl					:=0;
		down_valve_ctl				:=0;
		mv_alarm10007				:=1;
	END_IF
END_PROGRAM

(* POU CANOPEN_DATA/DATA_ACTIONG, ST *)
PROGRAM DATA_ACTIONG
VAR
END_VAR
can_encode_set();

anolog_in_out();
canopen_data_out();
digit_data_in();
END_PROGRAM

(* POU CANOPEN_DATA/can_encode_set, FBD *)
PROGRAM can_encode_set
VAR
	ENCOD_SET1: CAN1_SDO_WRITE;
	ENCOD_SET2: CAN1_SDO_WRITE;
	ENCOD_SET3: CAN1_SDO_WRITE;
	ENCOD_SET4: CAN1_SDO_WRITE;

	ENCOD_SET1_dat		:DWORD:=16#01000;
	ENCOD_SET2_dat		:DWORD:=16#200000;
	ENCOD_SET3_dat		:DWORD:=16#100000;
	ENCOD_SET4_dat		:DWORD:=16#65766173;
	ENCOD_SET9_dat		:DWORD:=16#64;

	ENCOD_SET5: CAN1_TRANSMIT;

	ENCOD_SET5_dat		: ARRAY [0..7] OF BYTE	:=1,0,0,0,0,0,0,0;	 (*启动*)
	ENCOD_SET6_dat		: ARRAY [0..7] OF BYTE	:=16#22,16#2,16#18,16#2,1,0,0,0;

	ENCOD_SET_dat1		: ARRAY [0..7] OF BYTE	:=16#2B,0,16#62,0,16#64,0,0,0;  (*循环周期*)
	ENCOD_SET_dat2		: ARRAY [0..7] OF BYTE	:=16#22,1,16#60,0,0,16#20,0,0;	 (*分辨率*)
	ENCOD_SET_dat5		: ARRAY [0..7] OF BYTE	:=16#22,2,16#60,0,16#0,16#0,16#0,16#02;	 (*总圈数*)
(*	ENCOD_SET_dat3		: ARRAY [0..7] OF BYTE	:=16#22,3,16#60,0,16#32,16#E3,16#FB,0;	 (*后四位 低到高 零点*)	*)
	ENCOD_SET_dat3		: ARRAY [0..7] OF BYTE	:=16#22,3,16#60,0,16#A8,16#44,16#E2,0;	 (*后四位 低到高 零点*)
	ENCOD_SET_dat30		: ARRAY [0..7] OF BYTE	:=16#22,16#17,16#10,0,16#E8,16#03,0,0;	 (*发状态*)
	ENCOD_SET_dat4		: ARRAY [0..7] OF BYTE	:=16#22,16#10,16#10,1,16#73,16#61,16#76,16#65;	 (*保存*)
	ENCOD_SET6			: CAN1_TRANSMIT;
	ENCOD_SET7			: CAN1_RECEIVE;
	DAT1						: ARRAY [0..7] OF BYTE;
	ENCOD_SET8			: CAN1_SDO_WRITE;
	ENCOD_SET7_dat		: DWORD:=16#1;
	ENCOD_SET9			: CAN1_SDO_WRITE;
	ENCOD_SET8_dat		: DWORD := 16#14;
	S1							:F_TRIG;
	encod_chg				: LSB_MSB_TO_DWORD;
	s2: BOOL;
	S3: TON;
	s4: BOOL;
	s5: BOOL;
	S6: R_TRIG;
	test1: FRAMWRITE;
	x2: BOOL;
	x3: BOOL;
	test2: FRAMREAD;
	test_button: BOOL;
	set1: BOOL;
END_VAR
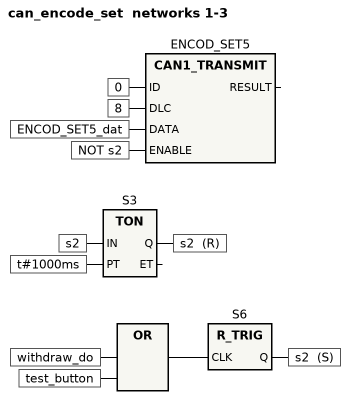
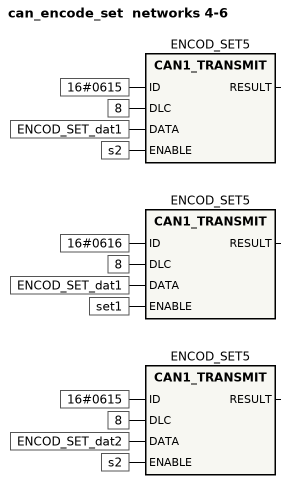
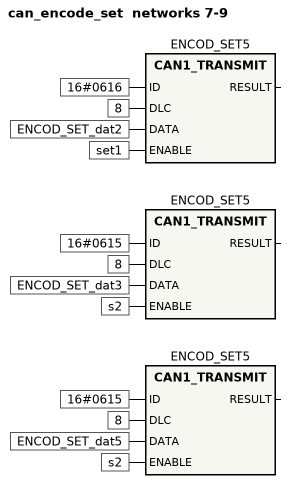
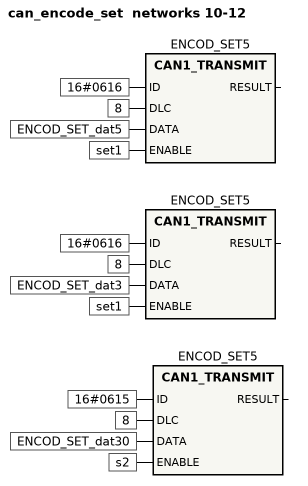
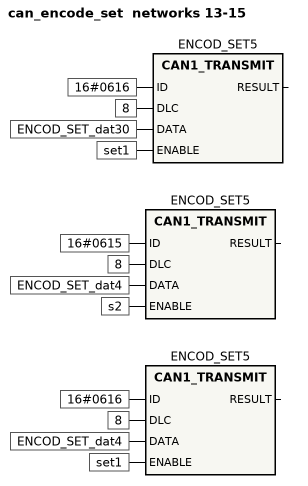
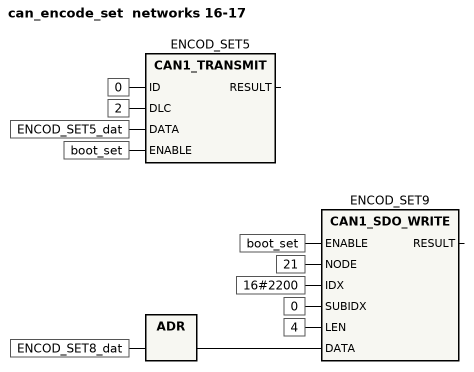
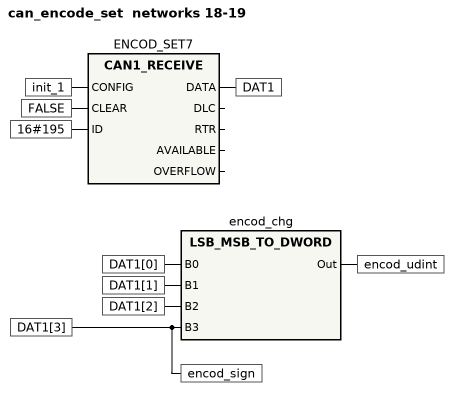
_FBD_ (* Function Block Diagram *)
NETWORK 1
	ENCOD_SET5:CAN1_TRANSMIT(ID: 0, DLC: 8, DATA: ENCOD_SET5_dat, ENABLE: NOT s2)
NETWORK 2
	S3:TON(IN: s2, PT: t#1000ms) => R s2
NETWORK 3
	S6:R_TRIG(CLK: OR(withdraw_do, test_button)) => S s2
NETWORK 4
	ENCOD_SET5:CAN1_TRANSMIT(ID: 16#0615, DLC: 8, DATA: ENCOD_SET_dat1, ENABLE: s2)
NETWORK 5
	ENCOD_SET5:CAN1_TRANSMIT(ID: 16#0616, DLC: 8, DATA: ENCOD_SET_dat1, ENABLE: set1)
NETWORK 6
	ENCOD_SET5:CAN1_TRANSMIT(ID: 16#0615, DLC: 8, DATA: ENCOD_SET_dat2, ENABLE: s2)
NETWORK 7
	ENCOD_SET5:CAN1_TRANSMIT(ID: 16#0616, DLC: 8, DATA: ENCOD_SET_dat2, ENABLE: set1)
NETWORK 8
	ENCOD_SET5:CAN1_TRANSMIT(ID: 16#0615, DLC: 8, DATA: ENCOD_SET_dat3, ENABLE: s2)
NETWORK 9
	ENCOD_SET5:CAN1_TRANSMIT(ID: 16#0615, DLC: 8, DATA: ENCOD_SET_dat5, ENABLE: s2)
NETWORK 10
	ENCOD_SET5:CAN1_TRANSMIT(ID: 16#0616, DLC: 8, DATA: ENCOD_SET_dat5, ENABLE: set1)
NETWORK 11
	ENCOD_SET5:CAN1_TRANSMIT(ID: 16#0616, DLC: 8, DATA: ENCOD_SET_dat3, ENABLE: set1)
NETWORK 12
	ENCOD_SET5:CAN1_TRANSMIT(ID: 16#0615, DLC: 8, DATA: ENCOD_SET_dat30, ENABLE: s2)
NETWORK 13
	ENCOD_SET5:CAN1_TRANSMIT(ID: 16#0616, DLC: 8, DATA: ENCOD_SET_dat30, ENABLE: set1)
NETWORK 14
	ENCOD_SET5:CAN1_TRANSMIT(ID: 16#0615, DLC: 8, DATA: ENCOD_SET_dat4, ENABLE: s2)
NETWORK 15
	ENCOD_SET5:CAN1_TRANSMIT(ID: 16#0616, DLC: 8, DATA: ENCOD_SET_dat4, ENABLE: set1)
NETWORK 16
	ENCOD_SET5:CAN1_TRANSMIT(ID: 0, DLC: 2, DATA: ENCOD_SET5_dat, ENABLE: boot_set)
NETWORK 17
	ENCOD_SET9:CAN1_SDO_WRITE(ENABLE: boot_set, NODE: 21, IDX: 16#2200, SUBIDX: 0, LEN: 4, DATA: ADR(ENCOD_SET8_dat))
NETWORK 18
	ENCOD_SET7:CAN1_RECEIVE(CONFIG: init_1, CLEAR: FALSE, ID: 16#195) => DAT1
NETWORK 19
	encod_chg:LSB_MSB_TO_DWORD(B0: DAT1[0], B1: DAT1[1], B2: DAT1[2], B3: <DAT1[3] => encod_sign>) => encod_udint
_END_FBD_
(* the same logic as Structured Text *)
(* Network 1 *)
ENCOD_SET5(ID := 0, DLC := 8, DATA := ENCOD_SET5_dat, ENABLE := NOT s2);
(* Network 2 *)
S3(IN := s2, PT := t#1000ms);
IF S3.Q THEN s2 := FALSE; END_IF;
(* Network 3 *)
S6(CLK := withdraw_do OR test_button);
IF S6.Q THEN s2 := TRUE; END_IF;
(* Network 4 *)
ENCOD_SET5(ID := 16#0615, DLC := 8, DATA := ENCOD_SET_dat1, ENABLE := s2);
(* Network 5 *)
ENCOD_SET5(ID := 16#0616, DLC := 8, DATA := ENCOD_SET_dat1, ENABLE := set1);
(* Network 6 *)
ENCOD_SET5(ID := 16#0615, DLC := 8, DATA := ENCOD_SET_dat2, ENABLE := s2);
(* Network 7 *)
ENCOD_SET5(ID := 16#0616, DLC := 8, DATA := ENCOD_SET_dat2, ENABLE := set1);
(* Network 8 *)
ENCOD_SET5(ID := 16#0615, DLC := 8, DATA := ENCOD_SET_dat3, ENABLE := s2);
(* Network 9 *)
ENCOD_SET5(ID := 16#0615, DLC := 8, DATA := ENCOD_SET_dat5, ENABLE := s2);
(* Network 10 *)
ENCOD_SET5(ID := 16#0616, DLC := 8, DATA := ENCOD_SET_dat5, ENABLE := set1);
(* Network 11 *)
ENCOD_SET5(ID := 16#0616, DLC := 8, DATA := ENCOD_SET_dat3, ENABLE := set1);
(* Network 12 *)
ENCOD_SET5(ID := 16#0615, DLC := 8, DATA := ENCOD_SET_dat30, ENABLE := s2);
(* Network 13 *)
ENCOD_SET5(ID := 16#0616, DLC := 8, DATA := ENCOD_SET_dat30, ENABLE := set1);
(* Network 14 *)
ENCOD_SET5(ID := 16#0615, DLC := 8, DATA := ENCOD_SET_dat4, ENABLE := s2);
(* Network 15 *)
ENCOD_SET5(ID := 16#0616, DLC := 8, DATA := ENCOD_SET_dat4, ENABLE := set1);
(* Network 16 *)
ENCOD_SET5(ID := 0, DLC := 2, DATA := ENCOD_SET5_dat, ENABLE := boot_set);
(* Network 17 *)
ENCOD_SET9(ENABLE := boot_set, NODE := 21, IDX := 16#2200, SUBIDX := 0, LEN := 4, DATA := ADR(ENCOD_SET8_dat));
(* Network 18 *)
ENCOD_SET7(CONFIG := init_1, CLEAR := FALSE, ID := 16#195);
DAT1 := ENCOD_SET7.DATA;
(* Network 19: see the listing above *)
END_PROGRAM

(* POU CANOPEN_DATA/LSB_MSB_TO_DWORD, ST *)
FUNCTION_BLOCK LSB_MSB_TO_DWORD
(* Converts 4 single bytes to a DWORD *)

VAR_INPUT
	B0: BYTE; (* LSB *)
	B1: BYTE;
	B2: BYTE;
	B3: BYTE; (* MSB *)
END_VAR

VAR_OUTPUT
	Out: DWORD;
END_VAR

VAR
	ptr: POINTER TO DWORD;
	Byte_IN: ARRAY[1..4] OF BYTE;
END_VAR
Byte_IN[1]:=B0;
Byte_IN[2]:=B1;
Byte_IN[3]:=B2;
Byte_IN[4]:=B3;

ptr:=ADR(Byte_IN);

Out:=ptr^;
END_FUNCTION_BLOCK

(* POU CANOPEN_DATA/anolog_in_out, ST *)
PROGRAM anolog_in_out
VAR

	water_h_temp		:WORD;
	foam_h_temp		:WORD;

	Analog_select		:WORD;

END_VAR
(****************************************************模拟数据上传值*********************************************************)
Analog_select		:=HighLowByteToWord(RX_id39[1],RX_id39[0]);


(******************************************水位标定值*********************************************)
IF water_low_sign_set 	THEN water_height_sign_L:=water_height_sign; 	END_IF
IF water_high_sign_set 	THEN water_height_sign_H:=water_height_sign; 	END_IF

(******************************************泡沫标定值********************************************)
IF foam_low_sign_set 	THEN foam_height_sign_L:=foam_height_sign; 	END_IF
IF foam_high_sign_set 	THEN foam_height_sign_H:=foam_height_sign; 	END_IF

(***************************************倾角传感器标定值****************************************)
IF down_zero_set THEN angle_x_offset:=angle_x;angle_y_offset:=angle_y;END_IF


(**************************************************模拟数据上传值*********************************************************)
CASE Analog_select OF
1:
	(****************************************水位标定值*******************************************)
	tx_id03[0]:=HighByteOfAWord(water_height_sign_L);
	tx_id03[1]:=LowByteOfAWord(water_height_sign_L);
	tx_id03[2]:=HighByteOfAWord(water_height_sign_H);
	tx_id03[3]:=LowByteOfAWord(water_height_sign_H);
	tx_id03[4]:=HighByteOfAWord(water_height_sign);
	tx_id03[5]:=LowByteOfAWord(water_height_sign);
5:
	(******************************************泡沫标定值********************************************)
	tx_id03[0]:=HighByteOfAWord(foam_height_sign_L);
	tx_id03[1]:=LowByteOfAWord(foam_height_sign_L);
	tx_id03[2]:=HighByteOfAWord(foam_height_sign_H);
	tx_id03[3]:=LowByteOfAWord(foam_height_sign_H);
	tx_id03[4]:=HighByteOfAWord(foam_height_sign);
	tx_id03[5]:=LowByteOfAWord(foam_height_sign);
6:
	(***************************************倾角传感器标定值****************************************)
	tx_id03[0]:=HighByteOfAWord(angle_x_offset);
	tx_id03[1]:=LowByteOfAWord(angle_x_offset);
	tx_id03[2]:=HighByteOfAWord(angle_y_offset);
	tx_id03[3]:=LowByteOfAWord(angle_y_offset);
	tx_id03[4]:=HighByteOfAWord(angle_x_m);
	tx_id03[5]:=LowByteOfAWord(angle_x_m);
	tx_id03[6]:=HighByteOfAWord(angle_y_m);
	tx_id03[7]:=LowByteOfAWord(angle_y_m);
ELSE
	tx_id03[0]:=0;
	tx_id03[1]:=0;
	tx_id03[2]:=0;
	tx_id03[3]:=0;
	tx_id03[4]:=0;
	tx_id03[5]:=0;
	tx_id03[6]:=0;
	tx_id03[7]:=0;

	tx_id04[0]:=0;
	tx_id04[1]:=0;
	tx_id04[2]:=0;
	tx_id04[3]:=0;
	tx_id04[4]:=0;
	tx_id04[5]:=0;
	tx_id04[6]:=0;
	tx_id04[7]:=0;
END_CASE



(**************************************垂直比例阀输出值****************************************)
tx_id05[0]:=HighByteOfAWord(left_front_desired_CR0032);
tx_id05[1]:=LowByteOfAWord(left_front_desired_CR0032);
tx_id05[2]:=HighByteOfAWord(left_back_desired_CR0032);
tx_id05[3]:=LowByteOfAWord(left_back_desired_CR0032);
tx_id05[4]:=HighByteOfAWord(right_front_desired_CR0032);
tx_id05[5]:=LowByteOfAWord(right_front_desired_CR0032);
tx_id05[6]:=HighByteOfAWord(right_back_desired_CR0032);
tx_id05[7]:=LowByteOfAWord(right_back_desired_CR0032);

(**************************************倾角传感器换算值****************************************)
tx_id06[0]:=HighByteOfAWord(angle_x);
tx_id06[1]:=LowByteOfAWord(angle_x);
tx_id06[2]:=HighByteOfAWord(angle_y);
tx_id06[3]:=LowByteOfAWord(angle_y);

(****************************************系统油温换算值*****************************************)

(****************************************系统油压换算值*****************************************)
tx_id07[2]:=HighByteOfAWord(oil_pressure);
tx_id07[3]:=LowByteOfAWord(oil_pressure);

(******************************************水位换算值*********************************************)
IF water_height_sign_H=water_height_sign_L 	THEN water_height_sign_H:=water_height_sign_L+1;														END_IF
water_h_temp:=REAL_TO_WORD(WORD_TO_REAL(water_height_sign-water_height_sign_L)/(water_height_sign_H-water_height_sign_L)*103);
IF water_h_temp<0  								THEN water_h_temp:=0;																						END_IF
IF water_h_temp>1000  							THEN water_h_temp:=0;																						END_IF
tx_id07[4]:=HighByteOfAWord(water_h_temp);
tx_id07[5]:=LowByteOfAWord(water_h_temp);

(*******************************************泡沫换算值********************************************)
IF foam_height_sign_H=foam_height_sign_L 	THEN foam_height_sign_H:=foam_height_sign_L+1;														END_IF
foam_h_temp:=REAL_TO_WORD(WORD_TO_REAL(foam_height_sign-foam_height_sign_L)/(foam_height_sign_H-foam_height_sign_L)*103);
IF foam_h_temp<0  								THEN foam_h_temp:=0;																						END_IF
IF foam_h_temp>1000  							THEN foam_h_temp:=0;																						END_IF
tx_id07[6]:=HighByteOfAWord(foam_h_temp);
tx_id07[7]:=LowByteOfAWord(foam_h_temp);

(*******************************************转速信号*********************************************)
tx_id08[0]:=HighByteOfAWord(REAL_TO_WORD(speed_m));
tx_id08[1]:=LowByteOfAWord(REAL_TO_WORD(speed_m));
END_PROGRAM

(* POU CANOPEN_DATA/HighLowByteToWord, ST *)
FUNCTION HighLowByteToWord : WORD
VAR_INPUT
	low	:	BYTE;
	high:	BYTE;
END_VAR
VAR
	hw1, hw2:WORD;
END_VAR
	(* produces a WORD out of LOW-BYTE and the High-Byte *)
	HighLowByteToWord := (BYTE_TO_WORD(low) OR SHL(  BYTE_TO_WORD(high),  8));

	HW1:=BYTE_TO_WORD(high);
	HW2:=SHL(  HW1,  8);
	HighLowByteToWord := (BYTE_TO_WORD(low) OR	HW2);
END_FUNCTION

(* POU CANOPEN_DATA/HighByteOfAWord, ST *)
FUNCTION HighByteOfAWord : BYTE
VAR_INPUT
	VarIn	:	WORD;
END_VAR
VAR
	HW1	:	WORD;

END_VAR
	(* liefert den HIGH-Teil des WORD als BYTE *)
	HW1:=SHR(VarIn,8);
	HighByteOfAWord :=WORD_TO_BYTE(HW1);
END_FUNCTION

(* POU CANOPEN_DATA/LowByteOfAWord, ST *)
FUNCTION LowByteOfAWord : BYTE
VAR_INPUT
	VarIn	:	WORD;
END_VAR
VAR
END_VAR
	(* liefert den LOW-Teil des WORD als BYTE *)
	LowByteOfAWord := WORD_TO_BYTE(VarIn);
END_FUNCTION

(* POU CANOPEN_DATA/canopen_data_out, FBD *)
PROGRAM canopen_data_out
VAR

END_VAR
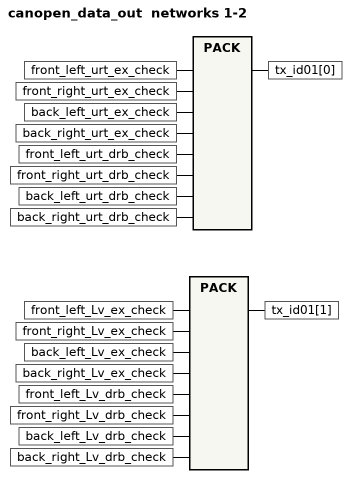
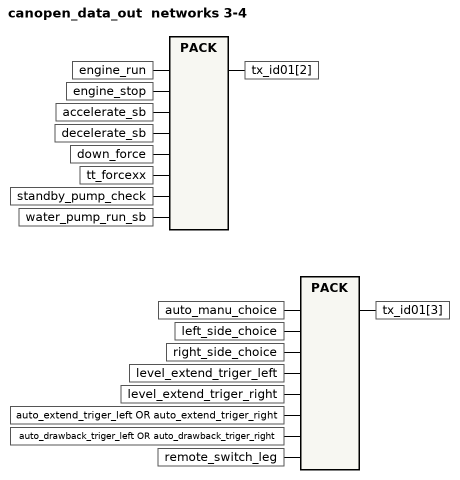
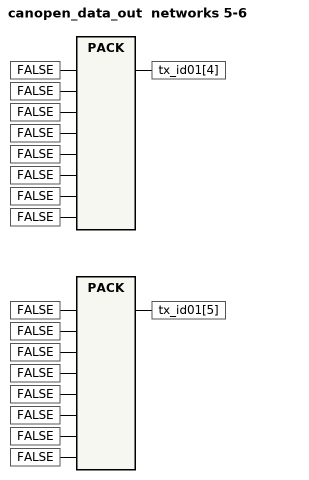
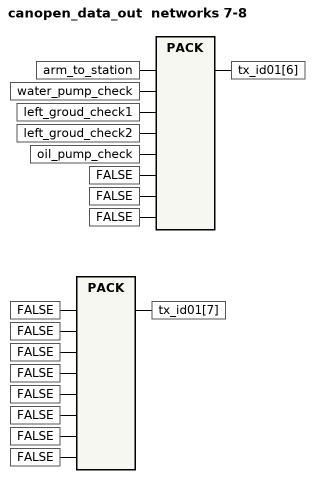
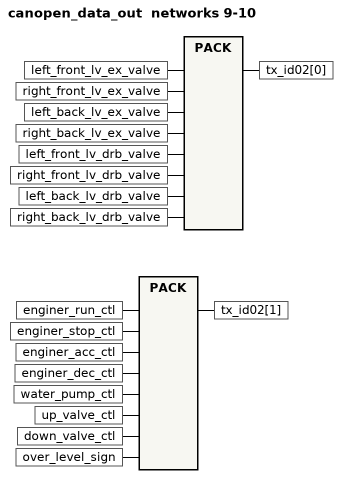
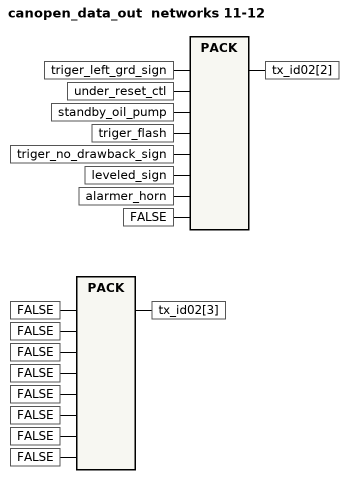
